LIN {X 0,Y 363.138,Z 659.015,A -85,B 0,C 180,E1 -13740.563,E2 -13740.563} C_VEL
LIN {X 0,Y 360.439,Z 673.892,A -85,B 0,C 180,E1 -13742.1,E2 -13742.1} C_VEL
LIN {X 0,Y 357.89,Z 687.3,A -85,B 0,C 180,E1 -13743.78,E2 -13743.78} C_VEL
LIN {X 0,Y 355.542,Z 698.752,A -85,B 0,C 180,E1 -13745.476,E2 -13745.476} C_VEL
LIN {X 0,Y 353.243,Z 710.279,A -85,B 0,C 180,E1 -13747.483,E2 -13747.483} C_VEL
LIN {X 0,Y 351.316,Z 720.192,A -85,B 0,C 180,E1 -13749.509,E2 -13749.509} C_VEL
LIN {X 0,Y 349.632,Z 729.753,A -85,B 0,C 180,E1 -13751.848,E2 -13751.848} C_VEL
LIN {X 0,Y 348.256,Z 737.796,A -85,B 0,C 180,E1 -13754.192,E2 -13754.192} C_VEL
LIN {X 0,Y 347.388,Z 744.678,A -85,B 0,C 180,E1 -13756.605,E2 -13756.605} C_VEL
LIN {X 0,Y 346.742,Z 750.015,A -85,B 0,C 180,E1 -13758.9,E2 -13758.9} C_VEL
LIN {X 0,Y 346.509,Z 753.412,A -85,B 0,C 180,E1 -13760.663,E2 -13760.663} C_VEL
LIN {X 0,Y 346.404,Z 757.9,A -85,B 0,C 180,E1 -13763.786,E2 -13763.786} C_VEL
LIN {X 0,Y 346.302,Z 760.292,A -85,B 0,C 180,E1 -13766.511,E2 -13766.511} C_VEL
LIN {X 0,Y 346.476,Z 761.273,A -85,B 0,C 180,E1 -13768.839,E2 -13768.839} C_VEL
LIN {X 0,Y 346.473,Z 761.269,A -85,B 0,C 180,E1 -13771.164,E2 -13771.164} C_VEL
LIN {X 0,Y 346.298,Z 760.218,A -85,B 0,C 180,E1 -13773.492,E2 -13773.492} C_VEL
LIN {X 0,Y 346.413,Z 758.208,A -85,B 0,C 180,E1 -13775.823,E2 -13775.823} C_VEL
LIN {X 0,Y 346.413,Z 755.082,A -85,B 0,C 180,E1 -13778.166,E2 -13778.166} C_VEL
LIN {X 0,Y 346.634,Z 750.942,A -85,B 0,C 180,E1 -13780.515,E2 -13780.515} C_VEL
LIN {X 0,Y 347.396,Z 744.256,A -85,B 0,C 180,E1 -13783.388,E2 -13783.388} C_VEL
LIN {X 0,Y 348.261,Z 737.113,A -85,B 0,C 180,E1 -13785.81,E2 -13785.81} C_VEL
LIN {X 0,Y 349.599,Z 728.749,A -85,B 0,C 180,E1 -13788.157,E2 -13788.157} C_VEL
LIN {X 0,Y 351.25,Z 718.757,A -85,B 0,C 180,E1 -13790.497,E2 -13790.497} C_VEL
LIN {X 0,Y 353.131,Z 708.481,A -85,B 0,C 180,E1 -13792.528,E2 -13792.528} C_VEL
LIN {X 0,Y 355.383,Z 696.336,A -85,B 0,C 180,E1 -13794.539,E2 -13794.539} C_VEL
LIN {X 0,Y 357.855,Z 682.977,A -85,B 0,C 180,E1 -13796.382,E2 -13796.382} C_VEL
LIN {X 0,Y 359.935,Z 670.909,A -85,B 0,C 180,E1 -13797.787,E2 -13797.787} C_VEL
LIN {X 0,Y 362.169,Z 656.954,A -85,B 0,C 180,E1 -13799.164,E2 -13799.164} C_VEL
LIN {X 0,Y 366.243,Z 636.712,A -85,B 0,C 180,E1 -13801.046,E2 -13801.046} C_VEL
LIN {X 0,Y 367.595,Z 629.602,A -85,B 0,C 180,E1 -13801.641,E2 -13801.641} C_VEL
LIN {X 0,Y 366.859,Z 616.235,A -85,B 0,C 180,E1 -13803.04,E2 -13803.04} C_VEL
LIN {X 0,Y 366.505,Z 599.284,A -85,B 0,C 180,E1 -13804.67,E2 -13804.67} C_VEL
LIN {X 0,Y 365.301,Z 587.346,A -85,B 0,C 180,E1 -13805.937,E2 -13805.937} C_VEL
LIN {X 0,Y 363.618,Z 576.417,A -85,B 0,C 180,E1 -13807.262,E2 -13807.262} C_VEL
LIN {X 0,Y 362.231,Z 569.674,A -85,B 0,C 180,E1 -13808.224,E2 -13808.224} C_VEL
LIN {X 0,Y 361.08,Z 564.227,A -85,B 0,C 180,E1 -13809.07,E2 -13809.07} C_VEL
LIN {X 0,Y 360.001,Z 559.824,A -85,B 0,C 180,E1 -13809.871,E2 -13809.871} C_VEL
LIN {X 0,Y 359.549,Z 557.218,A -85,B 0,C 180,E1 -13810.331,E2 -13810.331} C_VEL
LIN {X 0,Y 357.667,Z 548.632,A -85,B 0,C 180,E1 -13812.333,E2 -13812.333} C_VEL
LIN {X 0,Y 356.299,Z 544.697,A -85,B 0,C 180,E1 -13814.076,E2 -13814.076} C_VEL
LIN {X 0,Y 355.931,Z 542.529,A -85,B 0,C 180,E1 -13815.304,E2 -13815.304} C_VEL
LIN {X 0,Y 356.172,Z 540.509,A -85,B 0,C 180,E1 -13816.894,E2 -13816.894} C_VEL
LIN {X 0,Y 356.781,Z 539.56,A -85,B 0,C 180,E1 -13817.953,E2 -13817.953} C_VEL
LIN {X 0,Y 358.337,Z 540.28,A -85,B 0,C 180,E1 -13819.899,E2 -13819.899} C_VEL
LIN {X 0,Y 360.559,Z 541.255,A -85,B 0,C 180,E1 -13821.411,E2 -13821.411} C_VEL
LIN {X 0,Y 362.779,Z 542.718,A -85,B 0,C 180,E1 -13822.588,E2 -13822.588} C_VEL
LIN {X 0,Y 366.479,Z 546.75,A -85,B 0,C 180,E1 -13824.334,E2 -13824.334} C_VEL
LIN {X 0,Y 369.216,Z 550.249,A -85,B 0,C 180,E1 -13825.476,E2 -13825.476} C_VEL
LIN {X 0,Y 372.007,Z 554.619,A -85,B 0,C 180,E1 -13826.595,E2 -13826.595} C_VEL
LIN {X 0,Y 373.776,Z 559.648,A -85,B 0,C 180,E1 -13827.486,E2 -13827.486} C_VEL
LIN {X 0,Y 374.288,Z 561.573,A -85,B 0,C 180,E1 -13827.801,E2 -13827.801} C_VEL
LIN {X 0,Y 373.296,Z 567.896,A -85,B 0,C 180,E1 -13828.306,E2 -13828.306} C_VEL
LIN {X 0,Y 370.01,Z 584.666,A -85,B 0,C 180,E1 -13829.779,E2 -13829.779} C_VEL
LIN {X 0,Y 366.898,Z 599.707,A -85,B 0,C 180,E1 -13831.388,E2 -13831.388} C_VEL
LIN {X 0,Y 363.907,Z 613.147,A -85,B 0,C 180,E1 -13833.09,E2 -13833.09} C_VEL
LIN {X 0,Y 360.966,Z 625.629,A -85,B 0,C 180,E1 -13834.947,E2 -13834.947} C_VEL
LIN {X 0,Y 358.09,Z 637.94,A -85,B 0,C 180,E1 -13837.15,E2 -13837.15} C_VEL
LIN {X 0,Y 355.396,Z 648.703,A -85,B 0,C 180,E1 -13839.451,E2 -13839.451} C_VEL
LIN {X 0,Y 353.515,Z 656.559,A -85,B 0,C 180,E1 -13841.453,E2 -13841.453} C_VEL
LIN {X 0,Y 351.734,Z 664.142,A -85,B 0,C 180,E1 -13843.756,E2 -13843.756} C_VEL
LIN {X 0,Y 350.191,Z 670.343,A -85,B 0,C 180,E1 -13846.065,E2 -13846.065} C_VEL
LIN {X 0,Y 349.135,Z 675.359,A -85,B 0,C 180,E1 -13848.388,E2 -13848.388} C_VEL
LIN {X 0,Y 348.342,Z 679.303,A -85,B 0,C 180,E1 -13850.712,E2 -13850.712} C_VEL
LIN {X 0,Y 347.779,Z 682.101,A -85,B 0,C 180,E1 -13853.036,E2 -13853.036} C_VEL
LIN {X 0,Y 347.335,Z 683.994,A -85,B 0,C 180,E1 -13855.358,E2 -13855.358} C_VEL
LIN {X 0,Y 346.936,Z 684.871,A -85,B 0,C 180,E1 -13857.679,E2 -13857.679} C_VEL
LIN {X 0,Y 346.757,Z 684.777,A -85,B 0,C 180,E1 -13860.001,E2 -13860.001} C_VEL
LIN {X 0,Y 346.897,Z 683.694,A -85,B 0,C 180,E1 -13862.323,E2 -13862.323} C_VEL
LIN {X 0,Y 347.092,Z 681.603,A -85,B 0,C 180,E1 -13864.646,E2 -13864.646} C_VEL
LIN {X 0,Y 347.314,Z 678.062,A -85,B 0,C 180,E1 -13867.276,E2 -13867.276} C_VEL
LIN {X 0,Y 347.759,Z 673.198,A -85,B 0,C 180,E1 -13869.892,E2 -13869.892} C_VEL
LIN {X 0,Y 348.3,Z 667.576,A -85,B 0,C 180,E1 -13872.232,E2 -13872.232} C_VEL
LIN {X 0,Y 349.313,Z 660.704,A -85,B 0,C 180,E1 -13874.566,E2 -13874.566} C_VEL
LIN {X 0,Y 350.473,Z 652.438,A -85,B 0,C 180,E1 -13876.904,E2 -13876.904} C_VEL
LIN {X 0,Y 352.043,Z 642.556,A -85,B 0,C 180,E1 -13879.233,E2 -13879.233} C_VEL
LIN {X 0,Y 353.675,Z 632.321,A -85,B 0,C 180,E1 -13881.264,E2 -13881.264} C_VEL
LIN {X 0,Y 355.6,Z 620.344,A -85,B 0,C 180,E1 -13883.284,E2 -13883.284} C_VEL
LIN {X 0,Y 357.692,Z 607.625,A -85,B 0,C 180,E1 -13885.097,E2 -13885.097} C_VEL
LIN {X 0,Y 359.886,Z 593.111,A -85,B 0,C 180,E1 -13886.847,E2 -13886.847} C_VEL
LIN {X 0,Y 361.871,Z 579.208,A -85,B 0,C 180,E1 -13888.255,E2 -13888.255} C_VEL
LIN {X 0,Y 363.664,Z 565.161,A -85,B 0,C 180,E1 -13889.457,E2 -13889.457} C_VEL
LIN {X 0,Y 364.728,Z 556.813,A -85,B 0,C 180,E1 -13890.067,E2 -13890.067} C_VEL
LIN {X 0,Y 364.326,Z 554.698,A -85,B 0,C 180,E1 -13890.261,E2 -13890.261} C_VEL
LIN {X 0,Y 358.467,Z 539.997,A -85,B 0,C 180,E1 -13891.771,E2 -13891.771} C_VEL
LIN {X 0,Y 351.64,Z 524.321,A -85,B 0,C 180,E1 -13893.255,E2 -13893.255} C_VEL
LIN {X 0,Y 347.929,Z 516.364,A -85,B 0,C 180,E1 -13893.96,E2 -13893.96} C_VEL
LIN {X 0,Y 347.754,Z 515.48,A -85,B 0,C 180,E1 -13894.044,E2 -13894.044} C_VEL
LIN {X 0,Y 347.771,Z 515.479,A -85,B 0,C 180,E1 -13897.32,E2 -13897.32} C_VEL
LIN {X 0,Y 347.738,Z 515.483,A -85,B 0,C 180,E1 -13900.297,E2 -13900.297} C_VEL
LIN {X 0,Y 347.729,Z 515.483,A -85,B 0,C 180,E1 -13903.408,E2 -13903.408} C_VEL
LIN {X 0,Y 347.731,Z 515.482,A -85,B 0,C 180,E1 -13906.686,E2 -13906.686} C_VEL
LIN {X 0,Y 347.753,Z 515.482,A -85,B 0,C 180,E1 -13910.173,E2 -13910.173} C_VEL
LIN {X 0,Y 347.768,Z 515.478,A -85,B 0,C 180,E1 -13912.679,E2 -13912.679} C_VEL
LIN {X 0,Y 347.754,Z 515.485,A -85,B 0,C 180,E1 -13915.956,E2 -13915.956} C_VEL
LIN {X 0,Y 347.831,Z 515.679,A -85,B 0,C 180,E1 -13919.659,E2 -13919.659} C_VEL
LIN {X 0,Y 348.651,Z 519.993,A -85,B 0,C 180,E1 -13922.492,E2 -13922.492} C_VEL
LIN {X 0,Y 349.099,Z 524.824,A -85,B 0,C 180,E1 -13925.624,E2 -13925.624} C_VEL
LIN {X 0,Y 349.014,Z 529.788,A -85,B 0,C 180,E1 -13928.748,E2 -13928.748} C_VEL
LIN {X 0,Y 348.958,Z 531.353,A -85,B 0,C 180,E1 -13929.737,E2 -13929.737} C_VEL
LIN {X 0,Y 350.286,Z 534.706,A -85,B 0,C 180,E1 -13929.954,E2 -13929.954} C_VEL
LIN {X 0,Y 357.426,Z 551.292,A -85,B 0,C 180,E1 -13931.148,E2 -13931.148} C_VEL
LIN {X 0,Y 362.757,Z 565.923,A -85,B 0,C 180,E1 -13932.276,E2 -13932.276} C_VEL
LIN {X 0,Y 366.78,Z 578.552,A -85,B 0,C 180,E1 -13933.351,E2 -13933.351} C_VEL
LIN {X 0,Y 367.752,Z 582.268,A -85,B 0,C 180,E1 -13933.67,E2 -13933.67} C_VEL
LIN {X 0,Y 366.186,Z 596.258,A -85,B 0,C 180,E1 -13934.555,E2 -13934.555} C_VEL
LIN {X 0,Y 364.346,Z 610.122,A -85,B 0,C 180,E1 -13935.619,E2 -13935.619} C_VEL
LIN {X 0,Y 362.201,Z 624.446,A -85,B 0,C 180,E1 -13936.963,E2 -13936.963} C_VEL
LIN {X 0,Y 359.939,Z 637.66,A -85,B 0,C 180,E1 -13938.454,E2 -13938.454} C_VEL
LIN {X 0,Y 357.75,Z 649.93,A -85,B 0,C 180,E1 -13940.101,E2 -13940.101} C_VEL
LIN {X 0,Y 355.43,Z 662.146,A -85,B 0,C 180,E1 -13942.043,E2 -13942.043} C_VEL
LIN {X 0,Y 353.434,Z 672.571,A -85,B 0,C 180,E1 -13944.006,E2 -13944.006} C_VEL
LIN {X 0,Y 351.459,Z 682.629,A -85,B 0,C 180,E1 -13946.273,E2 -13946.273} C_VEL
LIN {X 0,Y 349.96,Z 690.122,A -85,B 0,C 180,E1 -13948.273,E2 -13948.273} C_VEL
LIN {X 0,Y 348.726,Z 697.402,A -85,B 0,C 180,E1 -13950.576,E2 -13950.576} C_VEL
LIN {X 0,Y 347.732,Z 703.363,A -85,B 0,C 180,E1 -13952.895,E2 -13952.895} C_VEL
LIN {X 0,Y 347.128,Z 708.203,A -85,B 0,C 180,E1 -13955.226,E2 -13955.226} C_VEL
LIN {X 0,Y 346.793,Z 711.131,A -85,B 0,C 180,E1 -13956.983,E2 -13956.983} C_VEL
LIN {X 0,Y 346.41,Z 714.204,A -85,B 0,C 180,E1 -13959.339,E2 -13959.339} C_VEL
LIN {X 0,Y 346.25,Z 716.196,A -85,B 0,C 180,E1 -13961.71,E2 -13961.71} C_VEL
LIN {X 0,Y 346.106,Z 717.28,A -85,B 0,C 180,E1 -13964.102,E2 -13964.102} C_VEL
LIN {X 0,Y 346.124,Z 717.343,A -85,B 0,C 180,E1 -13966.514,E2 -13966.514} C_VEL
LIN {X 0,Y 346.211,Z 716.409,A -85,B 0,C 180,E1 -13968.952,E2 -13968.952} C_VEL
LIN {X 0,Y 346.534,Z 714.459,A -85,B 0,C 180,E1 -13971.409,E2 -13971.409} C_VEL
LIN {X 0,Y 347.15,Z 710.676,A -85,B 0,C 180,E1 -13974.352,E2 -13974.352} C_VEL
LIN {X 0,Y 347.792,Z 707.099,A -85,B 0,C 180,E1 -13976.394,E2 -13976.394} C_VEL
LIN {X 0,Y 348.818,Z 701.582,A -85,B 0,C 180,E1 -13978.916,E2 -13978.916} C_VEL
LIN {X 0,Y 350.217,Z 694.579,A -85,B 0,C 180,E1 -13981.448,E2 -13981.448} C_VEL
LIN {X 0,Y 351.089,Z 690.641,A -85,B 0,C 180,E1 -13982.667,E2 -13982.667} C_VEL
LIN {X 0,Y 351.095,Z 687.889,A -85,B 0,C 180,E1 -13983.52,E2 -13983.52} C_VEL
LIN {X 0,Y 348.004,Z 678.593,A -85,B 0,C 180,E1 -13986.342,E2 -13986.342} C_VEL
LIN {X 0,Y 348.214,Z 675.241,A -85,B 0,C 180,E1 -13987.147,E2 -13987.147} C_VEL
LIN {X 0,Y 350.67,Z 665.25,A -85,B 0,C 180,E1 -13989.145,E2 -13989.145} C_VEL
LIN {X 0,Y 353.23,Z 654.18,A -85,B 0,C 180,E1 -13991.037,E2 -13991.037} C_VEL
LIN {X 0,Y 355.96,Z 642.094,A -85,B 0,C 180,E1 -13992.774,E2 -13992.774} C_VEL
LIN {X 0,Y 358.839,Z 628.158,A -85,B 0,C 180,E1 -13994.439,E2 -13994.439} C_VEL
LIN {X 0,Y 361.392,Z 614.482,A -85,B 0,C 180,E1 -13995.789,E2 -13995.789} C_VEL
LIN {X 0,Y 363.625,Z 600.382,A -85,B 0,C 180,E1 -13996.953,E2 -13996.953} C_VEL
LIN {X 0,Y 365.568,Z 586.338,A -85,B 0,C 180,E1 -13997.896,E2 -13997.896} C_VEL
LIN {X 0,Y 362.056,Z 574.059,A -85,B 0,C 180,E1 -13999.17,E2 -13999.17} C_VEL
LIN {X 0,Y 356.721,Z 560.139,A -85,B 0,C 180,E1 -14000.647,E2 -14000.647} C_VEL
LIN {X 0,Y 351.009,Z 548.123,A -85,B 0,C 180,E1 -14001.941,E2 -14001.941} C_VEL
LIN {X 0,Y 345.13,Z 537.197,A -85,B 0,C 180,E1 -14003.156,E2 -14003.156} C_VEL
LIN {X 0,Y 343.491,Z 534.071,A -85,B 0,C 180,E1 -14003.498,E2 -14003.498} C_VEL
LIN {X 0,Y 343.298,Z 533.359,A -85,B 0,C 180,E1 -14003.58,E2 -14003.58} C_VEL
LIN {X 0,Y 343.138,Z 529.364,A -85,B 0,C 180,E1 -14006.426,E2 -14006.426} C_VEL
LIN {X 0,Y 342.502,Z 525.206,A -85,B 0,C 180,E1 -14009.518,E2 -14009.518} C_VEL
LIN {X 0,Y 341.673,Z 520.486,A -85,B 0,C 180,E1 -14013.093,E2 -14013.093} C_VEL
LIN {X 0,Y 340.75,Z 516.352,A -85,B 0,C 180,E1 -14016.325,E2 -14016.325} C_VEL
LIN {X 0,Y 340.757,Z 516.352,A -85,B 0,C 180,E1 -14019.474,E2 -14019.474} C_VEL
LIN {X 0,Y 340.849,Z 516.341,A -85,B 0,C 180,E1 -14021.983,E2 -14021.983} C_VEL
LIN {X 0,Y 340.86,Z 516.334,A -85,B 0,C 180,E1 -14025.704,E2 -14025.704} C_VEL
LIN {X 0,Y 340.865,Z 516.331,A -85,B 0,C 180,E1 -14029.305,E2 -14029.305} C_VEL
LIN {X 0,Y 341.068,Z 516.31,A -85,B 0,C 180,E1 -14032.898,E2 -14032.898} C_VEL
LIN {X 0,Y 341.161,Z 516.296,A -85,B 0,C 180,E1 -14037.638,E2 -14037.638} C_VEL
LIN {X 0,Y 341.307,Z 516.284,A -85,B 0,C 180,E1 -14039.999,E2 -14039.999} C_VEL
LIN {X 0,Y 341.16,Z 516.293,A -85,B 0,C 180,E1 -14042.361,E2 -14042.361} C_VEL
LIN {X 0,Y 341.064,Z 516.312,A -85,B 0,C 180,E1 -14047.101,E2 -14047.101} C_VEL
LIN {X 0,Y 340.865,Z 516.337,A -85,B 0,C 180,E1 -14050.693,E2 -14050.693} C_VEL
LIN {X 0,Y 340.852,Z 516.339,A -85,B 0,C 180,E1 -14054.325,E2 -14054.325} C_VEL
LIN {X 0,Y 340.828,Z 516.3,A -85,B 0,C 180,E1 -14058.468,E2 -14058.468} C_VEL
LIN {X 0,Y 340.769,Z 516.347,A -85,B 0,C 180,E1 -14061.868,E2 -14061.868} C_VEL
LIN {X 0,Y 340.766,Z 516.315,A -85,B 0,C 180,E1 -14065.664,E2 -14065.664} C_VEL
LIN {X 0,Y 340.732,Z 516.355,A -85,B 0,C 180,E1 -14068.32,E2 -14068.32} C_VEL
LIN {X 0,Y 340.694,Z 516.359,A -85,B 0,C 180,E1 -14071.044,E2 -14071.044} C_VEL
LIN {X 0,Y 340.708,Z 516.454,A -85,B 0,C 180,E1 -14072.959,E2 -14072.959} C_VEL
LIN {X 0,Y 342.386,Z 523.899,A -85,B 0,C 180,E1 -14076.531,E2 -14076.531} C_VEL
LIN {X 0,Y 344.124,Z 531.611,A -85,B 0,C 180,E1 -14080.039,E2 -14080.039} C_VEL
LIN {X 0,Y 346.146,Z 541.37,A -85,B 0,C 180,E1 -14084.227,E2 -14084.227} C_VEL
LIN {X 0,Y 347.726,Z 549.268,A -85,B 0,C 180,E1 -14087.44,E2 -14087.44} C_VEL
LIN {X 0,Y 347.671,Z 553.507,A -85,B 0,C 180,E1 -14089.035,E2 -14089.035} C_VEL
LIN {X 0,Y 346.408,Z 563.412,A -85,B 0,C 180,E1 -14092.575,E2 -14092.575} C_VEL
LIN {X 0,Y 347.388,Z 567.065,A -85,B 0,C 180,E1 -14092.816,E2 -14092.816} C_VEL
LIN {X 0,Y 352.342,Z 581.881,A -85,B 0,C 180,E1 -14093.927,E2 -14093.927} C_VEL
LIN {X 0,Y 355.976,Z 596.537,A -85,B 0,C 180,E1 -14094.969,E2 -14094.969} C_VEL
LIN {X 0,Y 359.262,Z 613.763,A -85,B 0,C 180,E1 -14096.296,E2 -14096.296} C_VEL
LIN {X 0,Y 361.544,Z 630.3,A -85,B 0,C 180,E1 -14097.719,E2 -14097.719} C_VEL
LIN {X 0,Y 360.072,Z 641.655,A -85,B 0,C 180,E1 -14098.528,E2 -14098.528} C_VEL
LIN {X 0,Y 357.47,Z 656.478,A -85,B 0,C 180,E1 -14099.748,E2 -14099.748} C_VEL
LIN {X 0,Y 354.912,Z 670.176,A -85,B 0,C 180,E1 -14101.141,E2 -14101.141} C_VEL
LIN {X 0,Y 352.269,Z 683.008,A -85,B 0,C 180,E1 -14102.688,E2 -14102.688} C_VEL
LIN {X 0,Y 349.749,Z 695.417,A -85,B 0,C 180,E1 -14104.469,E2 -14104.469} C_VEL
LIN {X 0,Y 347.272,Z 707.025,A -85,B 0,C 180,E1 -14106.443,E2 -14106.443} C_VEL
LIN {X 0,Y 344.833,Z 718.604,A -85,B 0,C 180,E1 -14108.793,E2 -14108.793} C_VEL
LIN {X 0,Y 342.955,Z 728.348,A -85,B 0,C 180,E1 -14111.172,E2 -14111.172} C_VEL
LIN {X 0,Y 341.636,Z 735.634,A -85,B 0,C 180,E1 -14113.263,E2 -14113.263} C_VEL
LIN {X 0,Y 340.511,Z 743.379,A -85,B 0,C 180,E1 -14115.942,E2 -14115.942} C_VEL
LIN {X 0,Y 339.709,Z 749.641,A -85,B 0,C 180,E1 -14118.667,E2 -14118.667} C_VEL
LIN {X 0,Y 339.423,Z 753.021,A -85,B 0,C 180,E1 -14120.467,E2 -14120.467} C_VEL
LIN {X 0,Y 339.318,Z 756.502,A -85,B 0,C 180,E1 -14122.863,E2 -14122.863} C_VEL
LIN {X 0,Y 339.224,Z 759.021,A -85,B 0,C 180,E1 -14125.248,E2 -14125.248} C_VEL
LIN {X 0,Y 339.296,Z 760.457,A -85,B 0,C 180,E1 -14127.627,E2 -14127.627} C_VEL
LIN {X 0,Y 339.38,Z 760.964,A -85,B 0,C 180,E1 -14130.001,E2 -14130.001} C_VEL
LIN {X 0,Y 339.368,Z 760.397,A -85,B 0,C 180,E1 -14132.375,E2 -14132.375} C_VEL
LIN {X 0,Y 339.297,Z 758.874,A -85,B 0,C 180,E1 -14134.754,E2 -14134.754} C_VEL
LIN {X 0,Y 339.322,Z 756.269,A -85,B 0,C 180,E1 -14137.14,E2 -14137.14} C_VEL
LIN {X 0,Y 339.516,Z 751.522,A -85,B 0,C 180,E1 -14140.135,E2 -14140.135} C_VEL
LIN {X 0,Y 340.014,Z 746.466,A -85,B 0,C 180,E1 -14142.536,E2 -14142.536} C_VEL
LIN {X 0,Y 340.793,Z 740.198,A -85,B 0,C 180,E1 -14144.94,E2 -14144.94} C_VEL
LIN {X 0,Y 342.192,Z 731.492,A -85,B 0,C 180,E1 -14147.635,E2 -14147.635} C_VEL
LIN {X 0,Y 343.646,Z 722.545,A -85,B 0,C 180,E1 -14149.916,E2 -14149.916} C_VEL
LIN {X 0,Y 345.555,Z 712.361,A -85,B 0,C 180,E1 -14152.103,E2 -14152.103} C_VEL
LIN {X 0,Y 347.73,Z 701.327,A -85,B 0,C 180,E1 -14154.108,E2 -14154.108} C_VEL
LIN {X 0,Y 350.187,Z 688.648,A -85,B 0,C 180,E1 -14156.042,E2 -14156.042} C_VEL
LIN {X 0,Y 352.588,Z 675.091,A -85,B 0,C 180,E1 -14157.771,E2 -14157.771} C_VEL
LIN {X 0,Y 358.329,Z 646.316,A -85,B 0,C 180,E1 -14160.825,E2 -14160.825} C_VEL
LIN {X 0,Y 361.546,Z 630.746,A -85,B 0,C 180,E1 -14162.238,E2 -14162.238} C_VEL
LIN {X 0,Y 361.175,Z 617.764,A -85,B 0,C 180,E1 -14163.682,E2 -14163.682} C_VEL
LIN {X 0,Y 361.208,Z 601.756,A -85,B 0,C 180,E1 -14165.305,E2 -14165.305} C_VEL
LIN {X 0,Y 360.189,Z 588.151,A -85,B 0,C 180,E1 -14166.871,E2 -14166.871} C_VEL
LIN {X 0,Y 358.894,Z 578.855,A -85,B 0,C 180,E1 -14168.119,E2 -14168.119} C_VEL
LIN {X 0,Y 357.589,Z 570.516,A -85,B 0,C 180,E1 -14169.394,E2 -14169.394} C_VEL
LIN {X 0,Y 356.104,Z 562.093,A -85,B 0,C 180,E1 -14170.975,E2 -14170.975} C_VEL
LIN {X 0,Y 354.792,Z 554.339,A -85,B 0,C 180,E1 -14172.869,E2 -14172.869} C_VEL
LIN {X 0,Y 353.854,Z 551.132,A -85,B 0,C 180,E1 -14174.357,E2 -14174.357} C_VEL
LIN {X 0,Y 353.602,Z 548.557,A -85,B 0,C 180,E1 -14175.922,E2 -14175.922} C_VEL
LIN {X 0,Y 354.197,Z 546.683,A -85,B 0,C 180,E1 -14177.575,E2 -14177.575} C_VEL
LIN {X 0,Y 355.294,Z 546.707,A -85,B 0,C 180,E1 -14179.25,E2 -14179.25} C_VEL
LIN {X 0,Y 357.482,Z 547.514,A -85,B 0,C 180,E1 -14181.016,E2 -14181.016} C_VEL
LIN {X 0,Y 360.833,Z 550.296,A -85,B 0,C 180,E1 -14182.994,E2 -14182.994} C_VEL
LIN {X 0,Y 364.195,Z 554.214,A -85,B 0,C 180,E1 -14184.626,E2 -14184.626} C_VEL
LIN {X 0,Y 367.18,Z 558.764,A -85,B 0,C 180,E1 -14185.983,E2 -14185.983} C_VEL
LIN {X 0,Y 368.459,Z 561.71,A -85,B 0,C 180,E1 -14186.619,E2 -14186.619} C_VEL
LIN {X 0,Y 369.265,Z 565.365,A -85,B 0,C 180,E1 -14187.23,E2 -14187.23} C_VEL
LIN {X 0,Y 366.059,Z 580.597,A -85,B 0,C 180,E1 -14188.527,E2 -14188.527} C_VEL
LIN {X 0,Y 363.01,Z 594.419,A -85,B 0,C 180,E1 -14189.938,E2 -14189.938} C_VEL
LIN {X 0,Y 359.858,Z 607.979,A -85,B 0,C 180,E1 -14191.563,E2 -14191.563} C_VEL
LIN {X 0,Y 356.657,Z 620.811,A -85,B 0,C 180,E1 -14193.366,E2 -14193.366} C_VEL
LIN {X 0,Y 353.659,Z 632.613,A -85,B 0,C 180,E1 -14195.335,E2 -14195.335} C_VEL
LIN {X 0,Y 350.638,Z 644.102,A -85,B 0,C 180,E1 -14197.616,E2 -14197.616} C_VEL
LIN {X 0,Y 348.377,Z 652.718,A -85,B 0,C 180,E1 -14199.636,E2 -14199.636} C_VEL
LIN {X 0,Y 346.434,Z 660.061,A -85,B 0,C 180,E1 -14201.673,E2 -14201.673} C_VEL
LIN {X 0,Y 344.609,Z 667.128,A -85,B 0,C 180,E1 -14204.019,E2 -14204.019} C_VEL
LIN {X 0,Y 343.079,Z 672.996,A -85,B 0,C 180,E1 -14206.375,E2 -14206.375} C_VEL
LIN {X 0,Y 342.019,Z 677.625,A -85,B 0,C 180,E1 -14208.743,E2 -14208.743} C_VEL
LIN {X 0,Y 341.2,Z 681.494,A -85,B 0,C 180,E1 -14211.381,E2 -14211.381} C_VEL
LIN {X 0,Y 340.473,Z 684.179,A -85,B 0,C 180,E1 -14214.077,E2 -14214.077} C_VEL
LIN {X 0,Y 340.089,Z 685.513,A -85,B 0,C 180,E1 -14216.446,E2 -14216.446} C_VEL
LIN {X 0,Y 339.774,Z 685.809,A -85,B 0,C 180,E1 -14218.815,E2 -14218.815} C_VEL
LIN {X 0,Y 339.73,Z 685.179,A -85,B 0,C 180,E1 -14221.186,E2 -14221.186} C_VEL
LIN {X 0,Y 340.043,Z 683.494,A -85,B 0,C 180,E1 -14223.555,E2 -14223.555} C_VEL
LIN {X 0,Y 340.063,Z 680.87,A -85,B 0,C 180,E1 -14225.932,E2 -14225.932} C_VEL
LIN {X 0,Y 340.432,Z 677.2,A -85,B 0,C 180,E1 -14228.309,E2 -14228.309} C_VEL
LIN {X 0,Y 340.859,Z 672.382,A -85,B 0,C 180,E1 -14230.695,E2 -14230.695} C_VEL
LIN {X 0,Y 341.543,Z 666.42,A -85,B 0,C 180,E1 -14233.083,E2 -14233.083} C_VEL
LIN {X 0,Y 342.673,Z 659.135,A -85,B 0,C 180,E1 -14235.464,E2 -14235.464} C_VEL
LIN {X 0,Y 344.013,Z 650.33,A -85,B 0,C 180,E1 -14237.845,E2 -14237.845} C_VEL
LIN {X 0,Y 345.511,Z 641.257,A -85,B 0,C 180,E1 -14239.921,E2 -14239.921} C_VEL
LIN {X 0,Y 347.24,Z 630.713,A -85,B 0,C 180,E1 -14241.99,E2 -14241.99} C_VEL
LIN {X 0,Y 349.372,Z 618.351,A -85,B 0,C 180,E1 -14244.039,E2 -14244.039} C_VEL
LIN {X 0,Y 351.54,Z 605.148,A -85,B 0,C 180,E1 -14245.888,E2 -14245.888} C_VEL
LIN {X 0,Y 353.888,Z 590.046,A -85,B 0,C 180,E1 -14247.66,E2 -14247.66} C_VEL
LIN {X 0,Y 356.019,Z 575.397,A -85,B 0,C 180,E1 -14249.086,E2 -14249.086} C_VEL
LIN {X 0,Y 357.824,Z 560.818,A -85,B 0,C 180,E1 -14250.279,E2 -14250.279} C_VEL
LIN {X 0,Y 358.164,Z 558.328,A -85,B 0,C 180,E1 -14250.462,E2 -14250.462} C_VEL
LIN {X 0,Y 353.964,Z 546.899,A -85,B 0,C 180,E1 -14251.682,E2 -14251.682} C_VEL
LIN {X 0,Y 347.166,Z 530.919,A -85,B 0,C 180,E1 -14253.29,E2 -14253.29} C_VEL
LIN {X 0,Y 340.877,Z 517.276,A -85,B 0,C 180,E1 -14254.565,E2 -14254.565} C_VEL
LIN {X 0,Y 340.718,Z 516.359,A -85,B 0,C 180,E1 -14254.65,E2 -14254.65} C_VEL
LIN {X 0,Y 340.717,Z 516.356,A -85,B 0,C 180,E1 -14258.386,E2 -14258.386} C_VEL
LIN {X 0,Y 340.704,Z 516.359,A -85,B 0,C 180,E1 -14262.045,E2 -14262.045} C_VEL
LIN {X 0,Y 340.657,Z 516.365,A -85,B 0,C 180,E1 -14266.227,E2 -14266.227} C_VEL
LIN {X 0,Y 340.694,Z 516.36,A -85,B 0,C 180,E1 -14269.753,E2 -14269.753} C_VEL
LIN {X 0,Y 340.711,Z 516.357,A -85,B 0,C 180,E1 -14273.258,E2 -14273.258} C_VEL
LIN {X 0,Y 340.698,Z 516.365,A -85,B 0,C 180,E1 -14276.153,E2 -14276.153} C_VEL
LIN {X 0,Y 340.763,Z 516.532,A -85,B 0,C 180,E1 -14279.102,E2 -14279.102} C_VEL
LIN {X 0,Y 341.665,Z 521.168,A -85,B 0,C 180,E1 -14282.192,E2 -14282.192} C_VEL
LIN {X 0,Y 342.082,Z 524.974,A -85,B 0,C 180,E1 -14284.686,E2 -14284.686} C_VEL
LIN {X 0,Y 342.113,Z 529.503,A -85,B 0,C 180,E1 -14287.584,E2 -14287.584} C_VEL
LIN {X 0,Y 342.064,Z 531.756,A -85,B 0,C 180,E1 -14289.014,E2 -14289.014} C_VEL
LIN {X 0,Y 343.433,Z 535.172,A -85,B 0,C 180,E1 -14289.256,E2 -14289.256} C_VEL
LIN {X 0,Y 350.584,Z 551.695,A -85,B 0,C 180,E1 -14290.488,E2 -14290.488} C_VEL
LIN {X 0,Y 355.695,Z 565.542,A -85,B 0,C 180,E1 -14291.594,E2 -14291.594} C_VEL
LIN {X 0,Y 360.053,Z 578.984,A -85,B 0,C 180,E1 -14292.767,E2 -14292.767} C_VEL
LIN {X 0,Y 361.397,Z 583.652,A -85,B 0,C 180,E1 -14293.19,E2 -14293.19} C_VEL
LIN {X 0,Y 359.755,Z 597.908,A -85,B 0,C 180,E1 -14294.126,E2 -14294.126} C_VEL
LIN {X 0,Y 357.64,Z 613.036,A -85,B 0,C 180,E1 -14295.343,E2 -14295.343} C_VEL
LIN {X 0,Y 355.441,Z 626.988,A -85,B 0,C 180,E1 -14296.71,E2 -14296.71} C_VEL
LIN {X 0,Y 353.081,Z 639.967,A -85,B 0,C 180,E1 -14298.227,E2 -14298.227} C_VEL
LIN {X 0,Y 350.874,Z 651.931,A -85,B 0,C 180,E1 -14299.905,E2 -14299.905} C_VEL
LIN {X 0,Y 348.5,Z 663.904,A -85,B 0,C 180,E1 -14301.884,E2 -14301.884} C_VEL
LIN {X 0,Y 346.437,Z 674.197,A -85,B 0,C 180,E1 -14303.898,E2 -14303.898} C_VEL
LIN {X 0,Y 344.444,Z 684.073,A -85,B 0,C 180,E1 -14306.197,E2 -14306.197} C_VEL
LIN {X 0,Y 342.916,Z 691.396,A -85,B 0,C 180,E1 -14308.237,E2 -14308.237} C_VEL
LIN {X 0,Y 341.643,Z 698.514,A -85,B 0,C 180,E1 -14310.588,E2 -14310.588} C_VEL
LIN {X 0,Y 340.653,Z 704.399,A -85,B 0,C 180,E1 -14312.955,E2 -14312.955} C_VEL
LIN {X 0,Y 340.015,Z 709.096,A -85,B 0,C 180,E1 -14315.336,E2 -14315.336} C_VEL
LIN {X 0,Y 339.698,Z 711.954,A -85,B 0,C 180,E1 -14317.129,E2 -14317.129} C_VEL
LIN {X 0,Y 339.289,Z 714.894,A -85,B 0,C 180,E1 -14319.537,E2 -14319.537} C_VEL
LIN {X 0,Y 339.147,Z 716.821,A -85,B 0,C 180,E1 -14321.958,E2 -14321.958} C_VEL
LIN {X 0,Y 339.027,Z 717.769,A -85,B 0,C 180,E1 -14324.403,E2 -14324.403} C_VEL
LIN {X 0,Y 339.05,Z 717.769,A -85,B 0,C 180,E1 -14326.868,E2 -14326.868} C_VEL
LIN {X 0,Y 339.186,Z 716.695,A -85,B 0,C 180,E1 -14329.36,E2 -14329.36} C_VEL
LIN {X 0,Y 339.523,Z 714.641,A -85,B 0,C 180,E1 -14331.874,E2 -14331.874} C_VEL
LIN {X 0,Y 340.164,Z 711.113,A -85,B 0,C 180,E1 -14334.622,E2 -14334.622} C_VEL
LIN {X 0,Y 340.95,Z 707.01,A -85,B 0,C 180,E1 -14336.966,E2 -14336.966} C_VEL
LIN {X 0,Y 342.073,Z 701.349,A -85,B 0,C 180,E1 -14339.542,E2 -14339.542} C_VEL
LIN {X 0,Y 343.641,Z 694.244,A -85,B 0,C 180,E1 -14342.121,E2 -14342.121} C_VEL
LIN {X 0,Y 345.741,Z 685.467,A -85,B 0,C 180,E1 -14344.69,E2 -14344.69} C_VEL
LIN {X 0,Y 348.214,Z 675.241,A -85,B 0,C 180,E1 -14347.147,E2 -14347.147} C_VEL
LIN {X 0,Y 348.455,Z 671.831,A -85,B 0,C 180,E1 -14347.941,E2 -14347.941} C_VEL
LIN {X 0,Y 346.114,Z 660.483,A -85,B 0,C 180,E1 -14350.593,E2 -14350.593} C_VEL
LIN {X 0,Y 346.557,Z 656.521,A -85,B 0,C 180,E1 -14351.318,E2 -14351.318} C_VEL
LIN {X 0,Y 349.466,Z 644.29,A -85,B 0,C 180,E1 -14353.136,E2 -14353.136} C_VEL
LIN {X 0,Y 352.458,Z 630.465,A -85,B 0,C 180,E1 -14354.857,E2 -14354.857} C_VEL
LIN {X 0,Y 355.368,Z 615.865,A -85,B 0,C 180,E1 -14356.348,E2 -14356.348} C_VEL
LIN {X 0,Y 357.587,Z 602.695,A -85,B 0,C 180,E1 -14357.476,E2 -14357.476} C_VEL
LIN {X 0,Y 359.609,Z 587.963,A -85,B 0,C 180,E1 -14358.507,E2 -14358.507} C_VEL
LIN {X 0,Y 355.396,Z 573.834,A -85,B 0,C 180,E1 -14360.053,E2 -14360.053} C_VEL
LIN {X 0,Y 350.055,Z 560.252,A -85,B 0,C 180,E1 -14361.571,E2 -14361.571} C_VEL
LIN {X 0,Y 342.993,Z 545.87,A -85,B 0,C 180,E1 -14363.215,E2 -14363.215} C_VEL
LIN {X 0,Y 338.639,Z 538.042,A -85,B 0,C 180,E1 -14364.151,E2 -14364.151} C_VEL
LIN {X 0,Y 336.883,Z 535.201,A -85,B 0,C 180,E1 -14364.521,E2 -14364.521} C_VEL
LIN {X 0,Y 336.469,Z 533.841,A -85,B 0,C 180,E1 -14364.667,E2 -14364.667} C_VEL
LIN {X 0,Y 336.252,Z 530.568,A -85,B 0,C 180,E1 -14367.082,E2 -14367.082} C_VEL
LIN {X 0,Y 335.68,Z 526.957,A -85,B 0,C 180,E1 -14369.835,E2 -14369.835} C_VEL
LIN {X 0,Y 335.065,Z 523.467,A -85,B 0,C 180,E1 -14372.519,E2 -14372.519} C_VEL
LIN {X 0,Y 334.412,Z 520.133,A -85,B 0,C 180,E1 -14375.145,E2 -14375.145} C_VEL
LIN {X 0,Y 333.679,Z 517.235,A -85,B 0,C 180,E1 -14377.557,E2 -14377.557} C_VEL
LIN {X 0,Y 333.786,Z 517.217,A -85,B 0,C 180,E1 -14381.588,E2 -14381.588} C_VEL
LIN {X 0,Y 333.799,Z 517.214,A -85,B 0,C 180,E1 -14385.576,E2 -14385.576} C_VEL
LIN {X 0,Y 333.828,Z 517.207,A -85,B 0,C 180,E1 -14389.077,E2 -14389.077} C_VEL
LIN {X 0,Y 334.018,Z 517.186,A -85,B 0,C 180,E1 -14392.747,E2 -14392.747} C_VEL
LIN {X 0,Y 333.807,Z 517.209,A -85,B 0,C 180,E1 -14395.168,E2 -14395.168} C_VEL
LIN {X 0,Y 334.123,Z 517.173,A -85,B 0,C 180,E1 -14397.588,E2 -14397.588} C_VEL
LIN {X 0,Y 334.257,Z 517.163,A -85,B 0,C 180,E1 -14399.999,E2 -14399.999} C_VEL
LIN {X 0,Y 334.098,Z 517.172,A -85,B 0,C 180,E1 -14402.411,E2 -14402.411} C_VEL
LIN {X 0,Y 334.014,Z 517.191,A -85,B 0,C 180,E1 -14407.252,E2 -14407.252} C_VEL
LIN {X 0,Y 333.827,Z 517.213,A -85,B 0,C 180,E1 -14410.922,E2 -14410.922} C_VEL
LIN {X 0,Y 333.797,Z 517.216,A -85,B 0,C 180,E1 -14414.634,E2 -14414.634} C_VEL
LIN {X 0,Y 333.787,Z 517.177,A -85,B 0,C 180,E1 -14418.656,E2 -14418.656} C_VEL
LIN {X 0,Y 333.723,Z 517.216,A -85,B 0,C 180,E1 -14422.275,E2 -14422.275} C_VEL
LIN {X 0,Y 333.727,Z 517.201,A -85,B 0,C 180,E1 -14426.246,E2 -14426.246} C_VEL
LIN {X 0,Y 333.701,Z 517.232,A -85,B 0,C 180,E1 -14428.972,E2 -14428.972} C_VEL
LIN {X 0,Y 333.662,Z 517.35,A -85,B 0,C 180,E1 -14432.342,E2 -14432.342} C_VEL
LIN {X 0,Y 335.32,Z 524.667,A -85,B 0,C 180,E1 -14435.933,E2 -14435.933} C_VEL
LIN {X 0,Y 337.046,Z 532.368,A -85,B 0,C 180,E1 -14439.513,E2 -14439.513} C_VEL
LIN {X 0,Y 338.899,Z 541.365,A -85,B 0,C 180,E1 -14443.465,E2 -14443.465} C_VEL
LIN {X 0,Y 340.281,Z 548.106,A -85,B 0,C 180,E1 -14446.292,E2 -14446.292} C_VEL
LIN {X 0,Y 340.893,Z 552.154,A -85,B 0,C 180,E1 -14447.918,E2 -14447.918} C_VEL
LIN {X 0,Y 340.264,Z 558.251,A -85,B 0,C 180,E1 -14450.189,E2 -14450.189} C_VEL
LIN {X 0,Y 339.791,Z 562.191,A -85,B 0,C 180,E1 -14451.555,E2 -14451.555} C_VEL
LIN {X 0,Y 340.95,Z 566.07,A -85,B 0,C 180,E1 -14451.842,E2 -14451.842} C_VEL
LIN {X 0,Y 346.409,Z 582.721,A -85,B 0,C 180,E1 -14453.14,E2 -14453.14} C_VEL
LIN {X 0,Y 349.263,Z 593.517,A -85,B 0,C 180,E1 -14453.961,E2 -14453.961} C_VEL
LIN {X 0,Y 352.555,Z 610.412,A -85,B 0,C 180,E1 -14455.292,E2 -14455.292} C_VEL
LIN {X 0,Y 354.795,Z 626.575,A -85,B 0,C 180,E1 -14456.685,E2 -14456.685} C_VEL
LIN {X 0,Y 355.455,Z 633.074,A -85,B 0,C 180,E1 -14457.281,E2 -14457.281} C_VEL
LIN {X 0,Y 353.104,Z 647.27,A -85,B 0,C 180,E1 -14458.337,E2 -14458.337} C_VEL
LIN {X 0,Y 350.239,Z 662.244,A -85,B 0,C 180,E1 -14459.708,E2 -14459.708} C_VEL
LIN {X 0,Y 347.374,Z 676.296,A -85,B 0,C 180,E1 -14461.283,E2 -14461.283} C_VEL
LIN {X 0,Y 344.633,Z 689.192,A -85,B 0,C 180,E1 -14463.018,E2 -14463.018} C_VEL
LIN {X 0,Y 341.842,Z 701.615,A -85,B 0,C 180,E1 -14464.999,E2 -14464.999} C_VEL
LIN {X 0,Y 339.294,Z 712.902,A -85,B 0,C 180,E1 -14467.148,E2 -14467.148} C_VEL
LIN {X 0,Y 337.287,Z 722.206,A -85,B 0,C 180,E1 -14469.256,E2 -14469.256} C_VEL
LIN {X 0,Y 335.54,Z 731.317,A -85,B 0,C 180,E1 -14471.69,E2 -14471.69} C_VEL
LIN {X 0,Y 334.073,Z 738.999,A -85,B 0,C 180,E1 -14474.13,E2 -14474.13} C_VEL
LIN {X 0,Y 333.193,Z 745.294,A -85,B 0,C 180,E1 -14476.585,E2 -14476.585} C_VEL
LIN {X 0,Y 332.505,Z 750.447,A -85,B 0,C 180,E1 -14479.035,E2 -14479.035} C_VEL
LIN {X 0,Y 332.238,Z 754.491,A -85,B 0,C 180,E1 -14481.486,E2 -14481.486} C_VEL
LIN {X 0,Y 332.217,Z 757.463,A -85,B 0,C 180,E1 -14483.93,E2 -14483.93} C_VEL
LIN {X 0,Y 332.137,Z 759.439,A -85,B 0,C 180,E1 -14486.362,E2 -14486.362} C_VEL
LIN {X 0,Y 332.343,Z 760.382,A -85,B 0,C 180,E1 -14488.79,E2 -14488.79} C_VEL
LIN {X 0,Y 332.346,Z 760.361,A -85,B 0,C 180,E1 -14491.213,E2 -14491.213} C_VEL
LIN {X 0,Y 332.142,Z 759.266,A -85,B 0,C 180,E1 -14493.641,E2 -14493.641} C_VEL
LIN {X 0,Y 332.282,Z 757.059,A -85,B 0,C 180,E1 -14496.24,E2 -14496.24} C_VEL
LIN {X 0,Y 332.264,Z 754.055,A -85,B 0,C 180,E1 -14498.516,E2 -14498.516} C_VEL
LIN {X 0,Y 332.529,Z 749.865,A -85,B 0,C 180,E1 -14500.967,E2 -14500.967} C_VEL
LIN {X 0,Y 333.199,Z 744.444,A -85,B 0,C 180,E1 -14503.417,E2 -14503.417} C_VEL
LIN {X 0,Y 334.08,Z 737.783,A -85,B 0,C 180,E1 -14505.873,E2 -14505.873} C_VEL
LIN {X 0,Y 335.466,Z 729.771,A -85,B 0,C 180,E1 -14508.317,E2 -14508.317} C_VEL
LIN {X 0,Y 337.19,Z 720.136,A -85,B 0,C 180,E1 -14510.753,E2 -14510.753} C_VEL
LIN {X 0,Y 339.443,Z 708.609,A -85,B 0,C 180,E1 -14513.166,E2 -14513.166} C_VEL
LIN {X 0,Y 341.848,Z 696.73,A -85,B 0,C 180,E1 -14515.233,E2 -14515.233} C_VEL
LIN {X 0,Y 344.301,Z 684.566,A -85,B 0,C 180,E1 -14517.013,E2 -14517.013} C_VEL
LIN {X 0,Y 346.71,Z 671.682,A -85,B 0,C 180,E1 -14518.614,E2 -14518.614} C_VEL
LIN {X 0,Y 351.366,Z 651.047,A -85,B 0,C 180,E1 -14521.002,E2 -14521.002} C_VEL
LIN {X 0,Y 355.146,Z 635.262,A -85,B 0,C 180,E1 -14522.543,E2 -14522.543} C_VEL
LIN {X 0,Y 355.608,Z 633.039,A -85,B 0,C 180,E1 -14522.741,E2 -14522.741} C_VEL
LIN {X 0,Y 355.551,Z 619.845,A -85,B 0,C 180,E1 -14524.288,E2 -14524.288} C_VEL
LIN {X 0,Y 356.029,Z 604.246,A -85,B 0,C 180,E1 -14525.97,E2 -14525.97} C_VEL
LIN {X 0,Y 355.462,Z 591.655,A -85,B 0,C 180,E1 -14527.504,E2 -14527.504} C_VEL
LIN {X 0,Y 354.486,Z 581.867,A -85,B 0,C 180,E1 -14528.908,E2 -14528.908} C_VEL
LIN {X 0,Y 353.668,Z 574.442,A -85,B 0,C 180,E1 -14530.131,E2 -14530.131} C_VEL
LIN {X 0,Y 352.626,Z 566.818,A -85,B 0,C 180,E1 -14531.665,E2 -14531.665} C_VEL
LIN {X 0,Y 352.097,Z 561.344,A -85,B 0,C 180,E1 -14532.995,E2 -14532.995} C_VEL
LIN {X 0,Y 351.587,Z 558.857,A -85,B 0,C 180,E1 -14533.978,E2 -14533.978} C_VEL
LIN {X 0,Y 351.232,Z 555.165,A -85,B 0,C 180,E1 -14536.084,E2 -14536.084} C_VEL
LIN {X 0,Y 351.83,Z 553.394,A -85,B 0,C 180,E1 -14537.655,E2 -14537.655} C_VEL
LIN {X 0,Y 352.774,Z 553.332,A -85,B 0,C 180,E1 -14539.205,E2 -14539.205} C_VEL
LIN {X 0,Y 354.395,Z 553.935,A -85,B 0,C 180,E1 -14540.662,E2 -14540.662} C_VEL
LIN {X 0,Y 356.91,Z 555.812,A -85,B 0,C 180,E1 -14542.38,E2 -14542.38} C_VEL
LIN {X 0,Y 360.097,Z 559.53,A -85,B 0,C 180,E1 -14544.162,E2 -14544.162} C_VEL
LIN {X 0,Y 362.856,Z 563.77,A -85,B 0,C 180,E1 -14545.539,E2 -14545.539} C_VEL
LIN {X 0,Y 363.895,Z 566.229,A -85,B 0,C 180,E1 -14546.148,E2 -14546.148} C_VEL
LIN {X 0,Y 364.325,Z 568.043,A -85,B 0,C 180,E1 -14546.478,E2 -14546.478} C_VEL
LIN {X 0,Y 360.402,Z 585.49,A -85,B 0,C 180,E1 -14548.074,E2 -14548.074} C_VEL
LIN {X 0,Y 356.496,Z 601.3,A -85,B 0,C 180,E1 -14549.821,E2 -14549.821} C_VEL
LIN {X 0,Y 352.412,Z 616.982,A -85,B 0,C 180,E1 -14551.915,E2 -14551.915} C_VEL
LIN {X 0,Y 348.809,Z 630.056,A -85,B 0,C 180,E1 -14554.009,E2 -14554.009} C_VEL
LIN {X 0,Y 345.421,Z 642.306,A -85,B 0,C 180,E1 -14556.377,E2 -14556.377} C_VEL
LIN {X 0,Y 342.567,Z 652.097,A -85,B 0,C 180,E1 -14558.645,E2 -14558.645} C_VEL
LIN {X 0,Y 340.424,Z 659.654,A -85,B 0,C 180,E1 -14560.712,E2 -14560.712} C_VEL
LIN {X 0,Y 338.394,Z 666.958,A -85,B 0,C 180,E1 -14563.097,E2 -14563.097} C_VEL
LIN {X 0,Y 336.67,Z 672.973,A -85,B 0,C 180,E1 -14565.493,E2 -14565.493} C_VEL
LIN {X 0,Y 335.4,Z 677.778,A -85,B 0,C 180,E1 -14567.905,E2 -14567.905} C_VEL
LIN {X 0,Y 334.479,Z 681.545,A -85,B 0,C 180,E1 -14570.323,E2 -14570.323} C_VEL
LIN {X 0,Y 333.822,Z 684.209,A -85,B 0,C 180,E1 -14572.744,E2 -14572.744} C_VEL
LIN {X 0,Y 333.314,Z 685.933,A -85,B 0,C 180,E1 -14575.162,E2 -14575.162} C_VEL
LIN {X 0,Y 332.865,Z 686.698,A -85,B 0,C 180,E1 -14577.58,E2 -14577.58} C_VEL
LIN {X 0,Y 332.662,Z 686.44,A -85,B 0,C 180,E1 -14580.001,E2 -14580.001} C_VEL
LIN {X 0,Y 332.826,Z 685.245,A -85,B 0,C 180,E1 -14582.421,E2 -14582.421} C_VEL
LIN {X 0,Y 333.008,Z 682.988,A -85,B 0,C 180,E1 -14584.843,E2 -14584.843} C_VEL
LIN {X 0,Y 333.298,Z 679.131,A -85,B 0,C 180,E1 -14587.665,E2 -14587.665} C_VEL
LIN {X 0,Y 333.74,Z 674.203,A -85,B 0,C 180,E1 -14590.312,E2 -14590.312} C_VEL
LIN {X 0,Y 334.393,Z 668.444,A -85,B 0,C 180,E1 -14592.75,E2 -14592.75} C_VEL
LIN {X 0,Y 335.548,Z 660.828,A -85,B 0,C 180,E1 -14595.351,E2 -14595.351} C_VEL
LIN {X 0,Y 336.989,Z 651.688,A -85,B 0,C 180,E1 -14597.916,E2 -14597.916} C_VEL
LIN {X 0,Y 338.782,Z 641.311,A -85,B 0,C 180,E1 -14600.334,E2 -14600.334} C_VEL
LIN {X 0,Y 340.552,Z 630.623,A -85,B 0,C 180,E1 -14602.445,E2 -14602.445} C_VEL
LIN {X 0,Y 342.792,Z 618.107,A -85,B 0,C 180,E1 -14604.531,E2 -14604.531} C_VEL
LIN {X 0,Y 345.108,Z 604.491,A -85,B 0,C 180,E1 -14606.446,E2 -14606.446} C_VEL
LIN {X 0,Y 347.501,Z 589.473,A -85,B 0,C 180,E1 -14608.213,E2 -14608.213} C_VEL
LIN {X 0,Y 349.731,Z 574.674,A -85,B 0,C 180,E1 -14609.66,E2 -14609.66} C_VEL
LIN {X 0,Y 351.472,Z 559.585,A -85,B 0,C 180,E1 -14610.905,E2 -14610.905} C_VEL
LIN {X 0,Y 345.504,Z 544.333,A -85,B 0,C 180,E1 -14612.571,E2 -14612.571} C_VEL
LIN {X 0,Y 338.336,Z 527.856,A -85,B 0,C 180,E1 -14614.258,E2 -14614.258} C_VEL
LIN {X 0,Y 333.799,Z 517.935,A -85,B 0,C 180,E1 -14615.21,E2 -14615.21} C_VEL
LIN {X 0,Y 333.689,Z 517.232,A -85,B 0,C 180,E1 -14615.259,E2 -14615.259} C_VEL
LIN {X 0,Y 333.653,Z 517.238,A -85,B 0,C 180,E1 -14619.192,E2 -14619.192} C_VEL
LIN {X 0,Y 333.638,Z 517.239,A -85,B 0,C 180,E1 -14622.5,E2 -14622.5} C_VEL
LIN {X 0,Y 333.602,Z 517.245,A -85,B 0,C 180,E1 -14625.955,E2 -14625.955} C_VEL
LIN {X 0,Y 333.653,Z 517.237,A -85,B 0,C 180,E1 -14629.315,E2 -14629.315} C_VEL
LIN {X 0,Y 333.671,Z 517.233,A -85,B 0,C 180,E1 -14633.167,E2 -14633.167} C_VEL
LIN {X 0,Y 333.68,Z 517.234,A -85,B 0,C 180,E1 -14635.341,E2 -14635.341} C_VEL
LIN {X 0,Y 333.693,Z 517.373,A -85,B 0,C 180,E1 -14638.494,E2 -14638.494} C_VEL
LIN {X 0,Y 334.689,Z 522.355,A -85,B 0,C 180,E1 -14641.879,E2 -14641.879} C_VEL
LIN {X 0,Y 335.124,Z 526.165,A -85,B 0,C 180,E1 -14644.393,E2 -14644.393} C_VEL
LIN {X 0,Y 335.201,Z 530.634,A -85,B 0,C 180,E1 -14647.3,E2 -14647.3} C_VEL
LIN {X 0,Y 335.189,Z 532.163,A -85,B 0,C 180,E1 -14648.281,E2 -14648.281} C_VEL
LIN {X 0,Y 336.495,Z 535.509,A -85,B 0,C 180,E1 -14648.512,E2 -14648.512} C_VEL
LIN {X 0,Y 344.066,Z 552.82,A -85,B 0,C 180,E1 -14649.864,E2 -14649.864} C_VEL
LIN {X 0,Y 349.285,Z 566.914,A -85,B 0,C 180,E1 -14651.032,E2 -14651.032} C_VEL
LIN {X 0,Y 353.961,Z 581.72,A -85,B 0,C 180,E1 -14652.376,E2 -14652.376} C_VEL
LIN {X 0,Y 355.008,Z 585.459,A -85,B 0,C 180,E1 -14652.724,E2 -14652.724} C_VEL
LIN {X 0,Y 353.061,Z 601.44,A -85,B 0,C 180,E1 -14653.817,E2 -14653.817} C_VEL
LIN {X 0,Y 350.898,Z 615.969,A -85,B 0,C 180,E1 -14655.055,E2 -14655.055} C_VEL
LIN {X 0,Y 348.665,Z 629.468,A -85,B 0,C 180,E1 -14656.447,E2 -14656.447} C_VEL
LIN {X 0,Y 346.032,Z 643.192,A -85,B 0,C 180,E1 -14658.132,E2 -14658.132} C_VEL
LIN {X 0,Y 343.66,Z 655.72,A -85,B 0,C 180,E1 -14659.988,E2 -14659.988} C_VEL
LIN {X 0,Y 341.239,Z 667.216,A -85,B 0,C 180,E1 -14662.008,E2 -14662.008} C_VEL
LIN {X 0,Y 338.894,Z 678.289,A -85,B 0,C 180,E1 -14664.346,E2 -14664.346} C_VEL
LIN {X 0,Y 337.126,Z 686.515,A -85,B 0,C 180,E1 -14666.413,E2 -14666.413} C_VEL
LIN {X 0,Y 335.555,Z 694.534,A -85,B 0,C 180,E1 -14668.799,E2 -14668.799} C_VEL
LIN {X 0,Y 334.284,Z 701.193,A -85,B 0,C 180,E1 -14671.203,E2 -14671.203} C_VEL
LIN {X 0,Y 333.408,Z 706.621,A -85,B 0,C 180,E1 -14673.624,E2 -14673.624} C_VEL
LIN {X 0,Y 332.807,Z 711.016,A -85,B 0,C 180,E1 -14676.06,E2 -14676.06} C_VEL
LIN {X 0,Y 332.355,Z 714.297,A -85,B 0,C 180,E1 -14678.511,E2 -14678.511} C_VEL
LIN {X 0,Y 332.079,Z 716.638,A -85,B 0,C 180,E1 -14680.979,E2 -14680.979} C_VEL
LIN {X 0,Y 331.987,Z 717.965,A -85,B 0,C 180,E1 -14683.464,E2 -14683.464} C_VEL
LIN {X 0,Y 331.909,Z 718.331,A -85,B 0,C 180,E1 -14685.976,E2 -14685.976} C_VEL
LIN {X 0,Y 332.048,Z 717.71,A -85,B 0,C 180,E1 -14688.509,E2 -14688.509} C_VEL
LIN {X 0,Y 332.411,Z 715.62,A -85,B 0,C 180,E1 -14691.521,E2 -14691.521} C_VEL
LIN {X 0,Y 332.832,Z 713.298,A -85,B 0,C 180,E1 -14693.651,E2 -14693.651} C_VEL
LIN {X 0,Y 333.648,Z 709.363,A -85,B 0,C 180,E1 -14696.252,E2 -14696.252} C_VEL
LIN {X 0,Y 334.698,Z 704.189,A -85,B 0,C 180,E1 -14698.877,E2 -14698.877} C_VEL
LIN {X 0,Y 336.163,Z 697.667,A -85,B 0,C 180,E1 -14701.509,E2 -14701.509} C_VEL
LIN {X 0,Y 338.176,Z 689.606,A -85,B 0,C 180,E1 -14704.131,E2 -14704.131} C_VEL
LIN {X 0,Y 340.282,Z 681.348,A -85,B 0,C 180,E1 -14706.342,E2 -14706.342} C_VEL
LIN {X 0,Y 342.79,Z 671.611,A -85,B 0,C 180,E1 -14708.536,E2 -14708.536} C_VEL
LIN {X 0,Y 345.52,Z 660.717,A -85,B 0,C 180,E1 -14710.607,E2 -14710.607} C_VEL
LIN {X 0,Y 346.557,Z 656.521,A -85,B 0,C 180,E1 -14711.318,E2 -14711.318} C_VEL
LIN {X 0,Y 347.049,Z 652.502,A -85,B 0,C 180,E1 -14712.029,E2 -14712.029} C_VEL
LIN {X 0,Y 346.215,Z 646.035,A -85,B 0,C 180,E1 -14713.266,E2 -14713.266} C_VEL
LIN {X 0,Y 345.352,Z 639.224,A -85,B 0,C 180,E1 -14714.45,E2 -14714.45} C_VEL
LIN {X 0,Y 345.769,Z 634.67,A -85,B 0,C 180,E1 -14715.068,E2 -14715.068} C_VEL
LIN {X 0,Y 348.763,Z 620.539,A -85,B 0,C 180,E1 -14716.614,E2 -14716.614} C_VEL
LIN {X 0,Y 351.349,Z 606.17,A -85,B 0,C 180,E1 -14717.91,E2 -14717.91} C_VEL
LIN {X 0,Y 353.824,Z 590.51,A -85,B 0,C 180,E1 -14719.043,E2 -14719.043} C_VEL
LIN {X 0,Y 349.797,Z 576.656,A -85,B 0,C 180,E1 -14720.643,E2 -14720.643} C_VEL
LIN {X 0,Y 345.269,Z 564.706,A -85,B 0,C 180,E1 -14722.027,E2 -14722.027} C_VEL
LIN {X 0,Y 338.617,Z 550.565,A -85,B 0,C 180,E1 -14723.732,E2 -14723.732} C_VEL
LIN {X 0,Y 334.178,Z 542.519,A -85,B 0,C 180,E1 -14724.751,E2 -14724.751} C_VEL
LIN {X 0,Y 331.834,Z 538.559,A -85,B 0,C 180,E1 -14725.273,E2 -14725.273} C_VEL
LIN {X 0,Y 330.063,Z 535.664,A -85,B 0,C 180,E1 -14725.671,E2 -14725.671} C_VEL
LIN {X 0,Y 329.615,Z 534.359,A -85,B 0,C 180,E1 -14725.835,E2 -14725.835} C_VEL
LIN {X 0,Y 329.095,Z 529.999,A -85,B 0,C 180,E1 -14729.167,E2 -14729.167} C_VEL
LIN {X 0,Y 328.465,Z 526.543,A -85,B 0,C 180,E1 -14731.918,E2 -14731.918} C_VEL
LIN {X 0,Y 327.842,Z 523.183,A -85,B 0,C 180,E1 -14734.612,E2 -14734.612} C_VEL
LIN {X 0,Y 326.656,Z 518.12,A -85,B 0,C 180,E1 -14738.835,E2 -14738.835} C_VEL
LIN {X 0,Y 326.735,Z 518.094,A -85,B 0,C 180,E1 -14741.176,E2 -14741.176} C_VEL
LIN {X 0,Y 326.754,Z 518.093,A -85,B 0,C 180,E1 -14745.432,E2 -14745.432} C_VEL
LIN {X 0,Y 326.764,Z 518.087,A -85,B 0,C 180,E1 -14748.838,E2 -14748.838} C_VEL
LIN {X 0,Y 326.971,Z 518.062,A -85,B 0,C 180,E1 -14752.59,E2 -14752.59} C_VEL
LIN {X 0,Y 326.774,Z 518.085,A -85,B 0,C 180,E1 -14755.064,E2 -14755.064} C_VEL
LIN {X 0,Y 327.06,Z 518.053,A -85,B 0,C 180,E1 -14757.536,E2 -14757.536} C_VEL
LIN {X 0,Y 327.208,Z 518.041,A -85,B 0,C 180,E1 -14759.999,E2 -14759.999} C_VEL
LIN {X 0,Y 327.039,Z 518.052,A -85,B 0,C 180,E1 -14762.463,E2 -14762.463} C_VEL
LIN {X 0,Y 326.986,Z 518.057,A -85,B 0,C 180,E1 -14766.169,E2 -14766.169} C_VEL
LIN {X 0,Y 326.904,Z 518.065,A -85,B 0,C 180,E1 -14768.655,E2 -14768.655} C_VEL
LIN {X 0,Y 326.728,Z 518.086,A -85,B 0,C 180,E1 -14772.421,E2 -14772.421} C_VEL
LIN {X 0,Y 326.743,Z 518.09,A -85,B 0,C 180,E1 -14774.957,E2 -14774.957} C_VEL
LIN {X 0,Y 326.753,Z 518.055,A -85,B 0,C 180,E1 -14778.854,E2 -14778.854} C_VEL
LIN {X 0,Y 326.677,Z 518.08,A -85,B 0,C 180,E1 -14782.783,E2 -14782.783} C_VEL
LIN {X 0,Y 326.676,Z 518.093,A -85,B 0,C 180,E1 -14786.858,E2 -14786.858} C_VEL
LIN {X 0,Y 326.629,Z 518.112,A -85,B 0,C 180,E1 -14790.612,E2 -14790.612} C_VEL
LIN {X 0,Y 326.585,Z 518.12,A -85,B 0,C 180,E1 -14791.637,E2 -14791.637} C_VEL
LIN {X 0,Y 328.373,Z 525.986,A -85,B 0,C 180,E1 -14795.584,E2 -14795.584} C_VEL
LIN {X 0,Y 330.275,Z 534.63,A -85,B 0,C 180,E1 -14799.67,E2 -14799.67} C_VEL
LIN {X 0,Y 331.997,Z 542.9,A -85,B 0,C 180,E1 -14803.354,E2 -14803.354} C_VEL
LIN {X 0,Y 333.552,Z 550.607,A -85,B 0,C 180,E1 -14806.627,E2 -14806.627} C_VEL
LIN {X 0,Y 333.946,Z 554.184,A -85,B 0,C 180,E1 -14808.075,E2 -14808.075} C_VEL
LIN {X 0,Y 333.19,Z 560.49,A -85,B 0,C 180,E1 -14810.452,E2 -14810.452} C_VEL
LIN {X 0,Y 334.304,Z 564.493,A -85,B 0,C 180,E1 -14810.756,E2 -14810.756} C_VEL
LIN {X 0,Y 335.154,Z 566.806,A -85,B 0,C 180,E1 -14810.961,E2 -14810.961} C_VEL
LIN {X 0,Y 340.922,Z 584.505,A -85,B 0,C 180,E1 -14812.407,E2 -14812.407} C_VEL
LIN {X 0,Y 343.956,Z 596.924,A -85,B 0,C 180,E1 -14813.405,E2 -14813.405} C_VEL
LIN {X 0,Y 346.953,Z 613.337,A -85,B 0,C 180,E1 -14814.766,E2 -14814.766} C_VEL
LIN {X 0,Y 348.969,Z 629.818,A -85,B 0,C 180,E1 -14816.26,E2 -14816.26} C_VEL
LIN {X 0,Y 349.404,Z 633.723,A -85,B 0,C 180,E1 -14816.653,E2 -14816.653} C_VEL
LIN {X 0,Y 347.097,Z 647.64,A -85,B 0,C 180,E1 -14817.723,E2 -14817.723} C_VEL
LIN {X 0,Y 344.057,Z 662.813,A -85,B 0,C 180,E1 -14819.148,E2 -14819.148} C_VEL
LIN {X 0,Y 341.124,Z 676.388,A -85,B 0,C 180,E1 -14820.707,E2 -14820.707} C_VEL
LIN {X 0,Y 338.265,Z 689.179,A -85,B 0,C 180,E1 -14822.467,E2 -14822.467} C_VEL
LIN {X 0,Y 335.45,Z 701.109,A -85,B 0,C 180,E1 -14824.408,E2 -14824.408} C_VEL
LIN {X 0,Y 332.677,Z 712.742,A -85,B 0,C 180,E1 -14826.667,E2 -14826.667} C_VEL
LIN {X 0,Y 330.312,Z 723.035,A -85,B 0,C 180,E1 -14829.07,E2 -14829.07} C_VEL
LIN {X 0,Y 328.483,Z 732.079,A -85,B 0,C 180,E1 -14831.606,E2 -14831.606} C_VEL
LIN {X 0,Y 326.852,Z 740.336,A -85,B 0,C 180,E1 -14834.41,E2 -14834.41} C_VEL
LIN {X 0,Y 325.982,Z 746.372,A -85,B 0,C 180,E1 -14836.918,E2 -14836.918} C_VEL
LIN {X 0,Y 325.294,Z 752.254,A -85,B 0,C 180,E1 -14840.048,E2 -14840.048} C_VEL
LIN {X 0,Y 325.15,Z 755.7,A -85,B 0,C 180,E1 -14842.55,E2 -14842.55} C_VEL
LIN {X 0,Y 325.069,Z 758.173,A -85,B 0,C 180,E1 -14845.04,E2 -14845.04} C_VEL
LIN {X 0,Y 325.105,Z 759.586,A -85,B 0,C 180,E1 -14847.523,E2 -14847.523} C_VEL
LIN {X 0,Y 325.257,Z 760.052,A -85,B 0,C 180,E1 -14850.001,E2 -14850.001} C_VEL
LIN {X 0,Y 325.284,Z 759.905,A -85,B 0,C 180,E1 -14851.239,E2 -14851.239} C_VEL
LIN {X 0,Y 325.068,Z 758.784,A -85,B 0,C 180,E1 -14853.72,E2 -14853.72} C_VEL
LIN {X 0,Y 325.19,Z 756.737,A -85,B 0,C 180,E1 -14856.205,E2 -14856.205} C_VEL
LIN {X 0,Y 325.202,Z 753.528,A -85,B 0,C 180,E1 -14858.702,E2 -14858.702} C_VEL
LIN {X 0,Y 325.495,Z 749.304,A -85,B 0,C 180,E1 -14861.207,E2 -14861.207} C_VEL
LIN {X 0,Y 326.193,Z 743.865,A -85,B 0,C 180,E1 -14863.711,E2 -14863.711} C_VEL
LIN {X 0,Y 327.121,Z 737.169,A -85,B 0,C 180,E1 -14866.219,E2 -14866.219} C_VEL
LIN {X 0,Y 328.587,Z 729.118,A -85,B 0,C 180,E1 -14868.714,E2 -14868.714} C_VEL
LIN {X 0,Y 330.422,Z 719.449,A -85,B 0,C 180,E1 -14871.199,E2 -14871.199} C_VEL
LIN {X 0,Y 332.805,Z 707.865,A -85,B 0,C 180,E1 -14873.656,E2 -14873.656} C_VEL
LIN {X 0,Y 335.068,Z 696.949,A -85,B 0,C 180,E1 -14875.59,E2 -14875.59} C_VEL
LIN {X 0,Y 337.63,Z 684.758,A -85,B 0,C 180,E1 -14877.423,E2 -14877.423} C_VEL
LIN {X 0,Y 340.72,Z 670.32,A -85,B 0,C 180,E1 -14879.334,E2 -14879.334} C_VEL
LIN {X 0,Y 344.137,Z 656.783,A -85,B 0,C 180,E1 -14881.043,E2 -14881.043} C_VEL
LIN {X 0,Y 348.033,Z 641.5,A -85,B 0,C 180,E1 -14882.697,E2 -14882.697} C_VEL
LIN {X 0,Y 349.736,Z 634.469,A -85,B 0,C 180,E1 -14883.389,E2 -14883.389} C_VEL
LIN {X 0,Y 350.145,Z 620.664,A -85,B 0,C 180,E1 -14885.069,E2 -14885.069} C_VEL
LIN {X 0,Y 350.965,Z 605.862,A -85,B 0,C 180,E1 -14886.776,E2 -14886.776} C_VEL
LIN {X 0,Y 350.791,Z 594.432,A -85,B 0,C 180,E1 -14888.276,E2 -14888.276} C_VEL
LIN {X 0,Y 350.296,Z 585.936,A -85,B 0,C 180,E1 -14889.562,E2 -14889.562} C_VEL
LIN {X 0,Y 349.759,Z 578.47,A -85,B 0,C 180,E1 -14890.874,E2 -14890.874} C_VEL
LIN {X 0,Y 349.269,Z 571.722,A -85,B 0,C 180,E1 -14892.313,E2 -14892.313} C_VEL
LIN {X 0,Y 349.066,Z 566.884,A -85,B 0,C 180,E1 -14893.547,E2 -14893.547} C_VEL
LIN {X 0,Y 348.594,Z 563.508,A -85,B 0,C 180,E1 -14895.12,E2 -14895.12} C_VEL
LIN {X 0,Y 348.791,Z 561.114,A -85,B 0,C 180,E1 -14896.758,E2 -14896.758} C_VEL
LIN {X 0,Y 349.462,Z 559.932,A -85,B 0,C 180,E1 -14898.083,E2 -14898.083} C_VEL
LIN {X 0,Y 351.013,Z 560.259,A -85,B 0,C 180,E1 -14900.156,E2 -14900.156} C_VEL
LIN {X 0,Y 353.358,Z 561.73,A -85,B 0,C 180,E1 -14901.935,E2 -14901.935} C_VEL
LIN {X 0,Y 355.36,Z 563.94,A -85,B 0,C 180,E1 -14903.263,E2 -14903.263} C_VEL
LIN {X 0,Y 357.691,Z 567.328,A -85,B 0,C 180,E1 -14904.616,E2 -14904.616} C_VEL
LIN {X 0,Y 359.497,Z 570.976,A -85,B 0,C 180,E1 -14905.687,E2 -14905.687} C_VEL
LIN {X 0,Y 359.548,Z 571.924,A -85,B 0,C 180,E1 -14905.843,E2 -14905.843} C_VEL
LIN {X 0,Y 355,Z 589.507,A -85,B 0,C 180,E1 -14907.521,E2 -14907.521} C_VEL
LIN {X 0,Y 350.908,Z 604.662,A -85,B 0,C 180,E1 -14909.29,E2 -14909.29} C_VEL
LIN {X 0,Y 346.893,Z 618.708,A -85,B 0,C 180,E1 -14911.239,E2 -14911.239} C_VEL
LIN {X 0,Y 343.274,Z 630.832,A -85,B 0,C 180,E1 -14913.23,E2 -14913.23} C_VEL
LIN {X 0,Y 339.72,Z 642.688,A -85,B 0,C 180,E1 -14915.56,E2 -14915.56} C_VEL
LIN {X 0,Y 336.588,Z 652.766,A -85,B 0,C 180,E1 -14917.924,E2 -14917.924} C_VEL
LIN {X 0,Y 333.927,Z 661.271,A -85,B 0,C 180,E1 -14920.322,E2 -14920.322} C_VEL
LIN {X 0,Y 331.763,Z 668.441,A -85,B 0,C 180,E1 -14922.749,E2 -14922.749} C_VEL
LIN {X 0,Y 329.92,Z 674.353,A -85,B 0,C 180,E1 -14925.19,E2 -14925.19} C_VEL
LIN {X 0,Y 328.568,Z 679.035,A -85,B 0,C 180,E1 -14927.65,E2 -14927.65} C_VEL
LIN {X 0,Y 327.554,Z 682.691,A -85,B 0,C 180,E1 -14930.117,E2 -14930.117} C_VEL
LIN {X 0,Y 326.867,Z 685.296,A -85,B 0,C 180,E1 -14932.588,E2 -14932.588} C_VEL
LIN {X 0,Y 326.307,Z 686.909,A -85,B 0,C 180,E1 -14935.058,E2 -14935.058} C_VEL
LIN {X 0,Y 325.831,Z 687.621,A -85,B 0,C 180,E1 -14937.528,E2 -14937.528} C_VEL
LIN {X 0,Y 325.616,Z 687.28,A -85,B 0,C 180,E1 -14940.001,E2 -14940.001} C_VEL
LIN {X 0,Y 325.792,Z 685.996,A -85,B 0,C 180,E1 -14942.473,E2 -14942.473} C_VEL
LIN {X 0,Y 325.978,Z 684.949,A -85,B 0,C 180,E1 -14943.709,E2 -14943.709} C_VEL
LIN {X 0,Y 325.97,Z 682.147,A -85,B 0,C 180,E1 -14946.189,E2 -14946.189} C_VEL
LIN {X 0,Y 326.387,Z 678.331,A -85,B 0,C 180,E1 -14948.67,E2 -14948.67} C_VEL
LIN {X 0,Y 326.874,Z 673.325,A -85,B 0,C 180,E1 -14951.158,E2 -14951.158} C_VEL
LIN {X 0,Y 327.684,Z 667.142,A -85,B 0,C 180,E1 -14953.647,E2 -14953.647} C_VEL
LIN {X 0,Y 328.895,Z 659.647,A -85,B 0,C 180,E1 -14956.129,E2 -14956.129} C_VEL
LIN {X 0,Y 330.396,Z 650.65,A -85,B 0,C 180,E1 -14958.607,E2 -14958.607} C_VEL
LIN {X 0,Y 332.293,Z 639.894,A -85,B 0,C 180,E1 -14961.073,E2 -14961.073} C_VEL
LIN {X 0,Y 334.198,Z 628.783,A -85,B 0,C 180,E1 -14963.223,E2 -14963.223} C_VEL
LIN {X 0,Y 336.563,Z 615.774,A -85,B 0,C 180,E1 -14965.346,E2 -14965.346} C_VEL
LIN {X 0,Y 338.837,Z 602.697,A -85,B 0,C 180,E1 -14967.15,E2 -14967.15} C_VEL
LIN {X 0,Y 341.064,Z 588.673,A -85,B 0,C 180,E1 -14968.795,E2 -14968.795} C_VEL
LIN {X 0,Y 343.485,Z 573.653,A -85,B 0,C 180,E1 -14970.256,E2 -14970.256} C_VEL
LIN {X 0,Y 344.972,Z 561.853,A -85,B 0,C 180,E1 -14971.237,E2 -14971.237} C_VEL
LIN {X 0,Y 339.169,Z 546.932,A -85,B 0,C 180,E1 -14972.942,E2 -14972.942} C_VEL
LIN {X 0,Y 332.459,Z 531.291,A -85,B 0,C 180,E1 -14974.614,E2 -14974.614} C_VEL
LIN {X 0,Y 326.743,Z 518.688,A -85,B 0,C 180,E1 -14975.851,E2 -14975.851} C_VEL
LIN {X 0,Y 326.642,Z 518.112,A -85,B 0,C 180,E1 -14975.895,E2 -14975.895} C_VEL
LIN {X 0,Y 326.618,Z 518.114,A -85,B 0,C 180,E1 -14979.227,E2 -14979.227} C_VEL
LIN {X 0,Y 326.581,Z 518.119,A -85,B 0,C 180,E1 -14982.972,E2 -14982.972} C_VEL
LIN {X 0,Y 326.582,Z 518.117,A -85,B 0,C 180,E1 -14987.028,E2 -14987.028} C_VEL
LIN {X 0,Y 326.617,Z 518.114,A -85,B 0,C 180,E1 -14990.773,E2 -14990.773} C_VEL
LIN {X 0,Y 326.619,Z 518.117,A -85,B 0,C 180,E1 -14994.48,E2 -14994.48} C_VEL
LIN {X 0,Y 326.611,Z 518.168,A -85,B 0,C 180,E1 -14997.82,E2 -14997.82} C_VEL
LIN {X 0,Y 327.391,Z 521.954,A -85,B 0,C 180,E1 -15000.413,E2 -15000.413} C_VEL
LIN {X 0,Y 328.075,Z 526.113,A -85,B 0,C 180,E1 -15003.264,E2 -15003.264} C_VEL
LIN {X 0,Y 328.322,Z 530.259,A -85,B 0,C 180,E1 -15006.001,E2 -15006.001} C_VEL
LIN {X 0,Y 328.271,Z 532.545,A -85,B 0,C 180,E1 -15007.488,E2 -15007.488} C_VEL
LIN {X 0,Y 329.579,Z 535.827,A -85,B 0,C 180,E1 -15007.738,E2 -15007.738} C_VEL
LIN {X 0,Y 337.033,Z 552.571,A -85,B 0,C 180,E1 -15009.102,E2 -15009.102} C_VEL
LIN {X 0,Y 343.003,Z 568.587,A -85,B 0,C 180,E1 -15010.481,E2 -15010.481} C_VEL
LIN {X 0,Y 347.8,Z 584.057,A -85,B 0,C 180,E1 -15011.937,E2 -15011.937} C_VEL
LIN {X 0,Y 348.687,Z 587.404,A -85,B 0,C 180,E1 -15012.268,E2 -15012.268} C_VEL
LIN {X 0,Y 346.737,Z 602.466,A -85,B 0,C 180,E1 -15013.321,E2 -15013.321} C_VEL
LIN {X 0,Y 344.417,Z 617.326,A -85,B 0,C 180,E1 -15014.616,E2 -15014.616} C_VEL
LIN {X 0,Y 342.125,Z 630.667,A -85,B 0,C 180,E1 -15016.031,E2 -15016.031} C_VEL
LIN {X 0,Y 339.4,Z 644.28,A -85,B 0,C 180,E1 -15017.745,E2 -15017.745} C_VEL
LIN {X 0,Y 337.129,Z 655.857,A -85,B 0,C 180,E1 -15019.489,E2 -15019.489} C_VEL
LIN {X 0,Y 334.645,Z 667.381,A -85,B 0,C 180,E1 -15021.545,E2 -15021.545} C_VEL
LIN {X 0,Y 332.184,Z 678.505,A -85,B 0,C 180,E1 -15023.926,E2 -15023.926} C_VEL
LIN {X 0,Y 330.092,Z 687.856,A -85,B 0,C 180,E1 -15026.337,E2 -15026.337} C_VEL
LIN {X 0,Y 328.481,Z 695.708,A -85,B 0,C 180,E1 -15028.773,E2 -15028.773} C_VEL
LIN {X 0,Y 327.202,Z 702.283,A -85,B 0,C 180,E1 -15031.229,E2 -15031.229} C_VEL
LIN {X 0,Y 326.165,Z 708.773,A -85,B 0,C 180,E1 -15034.324,E2 -15034.324} C_VEL
LIN {X 0,Y 325.46,Z 713.596,A -85,B 0,C 180,E1 -15037.443,E2 -15037.443} C_VEL
LIN {X 0,Y 325.096,Z 716.265,A -85,B 0,C 180,E1 -15039.958,E2 -15039.958} C_VEL
LIN {X 0,Y 324.957,Z 718.022,A -85,B 0,C 180,E1 -15042.489,E2 -15042.489} C_VEL
LIN {X 0,Y 324.855,Z 718.752,A -85,B 0,C 180,E1 -15045.045,E2 -15045.045} C_VEL
LIN {X 0,Y 324.978,Z 718.422,A -85,B 0,C 180,E1 -15047.907,E2 -15047.907} C_VEL
LIN {X 0,Y 325.115,Z 717.279,A -85,B 0,C 180,E1 -15050.233,E2 -15050.233} C_VEL
LIN {X 0,Y 325.575,Z 714.941,A -85,B 0,C 180,E1 -15052.863,E2 -15052.863} C_VEL
LIN {X 0,Y 326.311,Z 711.537,A -85,B 0,C 180,E1 -15055.514,E2 -15055.514} C_VEL
LIN {X 0,Y 327.433,Z 706.537,A -85,B 0,C 180,E1 -15058.354,E2 -15058.354} C_VEL
LIN {X 0,Y 328.988,Z 699.818,A -85,B 0,C 180,E1 -15061.294,E2 -15061.294} C_VEL
LIN {X 0,Y 330.641,Z 693.438,A -85,B 0,C 180,E1 -15063.547,E2 -15063.547} C_VEL
LIN {X 0,Y 332.748,Z 685.605,A -85,B 0,C 180,E1 -15065.879,E2 -15065.879} C_VEL
LIN {X 0,Y 335.307,Z 676.207,A -85,B 0,C 180,E1 -15068.191,E2 -15068.191} C_VEL
LIN {X 0,Y 337.859,Z 666.776,A -85,B 0,C 180,E1 -15070.152,E2 -15070.152} C_VEL
LIN {X 0,Y 340.548,Z 656.369,A -85,B 0,C 180,E1 -15072.016,E2 -15072.016} C_VEL
LIN {X 0,Y 343.557,Z 644.048,A -85,B 0,C 180,E1 -15073.863,E2 -15073.863} C_VEL
LIN {X 0,Y 345.769,Z 634.67,A -85,B 0,C 180,E1 -15075.068,E2 -15075.068} C_VEL
LIN {X 0,Y 346.21,Z 630.081,A -85,B 0,C 180,E1 -15075.671,E2 -15075.671} C_VEL
LIN {X 0,Y 344.681,Z 615.043,A -85,B 0,C 180,E1 -15077.809,E2 -15077.809} C_VEL
LIN {X 0,Y 345.048,Z 610.043,A -85,B 0,C 180,E1 -15078.325,E2 -15078.325} C_VEL
LIN {X 0,Y 347.654,Z 595.016,A -85,B 0,C 180,E1 -15079.492,E2 -15079.492} C_VEL
LIN {X 0,Y 347.846,Z 592.076,A -85,B 0,C 180,E1 -15079.718,E2 -15079.718} C_VEL
LIN {X 0,Y 344.127,Z 579.178,A -85,B 0,C 180,E1 -15081.284,E2 -15081.284} C_VEL
LIN {X 0,Y 339.41,Z 566.573,A -85,B 0,C 180,E1 -15082.816,E2 -15082.816} C_VEL
LIN {X 0,Y 332.991,Z 552.765,A -85,B 0,C 180,E1 -15084.572,E2 -15084.572} C_VEL
LIN {X 0,Y 327.614,Z 543.264,A -85,B 0,C 180,E1 -15085.867,E2 -15085.867} C_VEL
LIN {X 0,Y 325.19,Z 539.293,A -85,B 0,C 180,E1 -15086.433,E2 -15086.433} C_VEL
LIN {X 0,Y 323.083,Z 536.07,A -85,B 0,C 180,E1 -15086.931,E2 -15086.931} C_VEL
LIN {X 0,Y 322.672,Z 534.887,A -85,B 0,C 180,E1 -15087.099,E2 -15087.099} C_VEL
LIN {X 0,Y 321.969,Z 530.202,A -85,B 0,C 180,E1 -15090.82,E2 -15090.82} C_VEL
LIN {X 0,Y 321.296,Z 526.247,A -85,B 0,C 180,E1 -15094.056,E2 -15094.056} C_VEL
LIN {X 0,Y 320.208,Z 521.524,A -85,B 0,C 180,E1 -15098.091,E2 -15098.091} C_VEL
LIN {X 0,Y 319.625,Z 518.983,A -85,B 0,C 180,E1 -15100.407,E2 -15100.407} C_VEL
LIN {X 0,Y 319.664,Z 518.973,A -85,B 0,C 180,E1 -15103.392,E2 -15103.392} C_VEL
LIN {X 0,Y 319.723,Z 518.965,A -85,B 0,C 180,E1 -15106.007,E2 -15106.007} C_VEL
LIN {X 0,Y 319.75,Z 518.965,A -85,B 0,C 180,E1 -15109.872,E2 -15109.872} C_VEL
LIN {X 0,Y 319.925,Z 518.939,A -85,B 0,C 180,E1 -15112.425,E2 -15112.425} C_VEL
LIN {X 0,Y 319.743,Z 518.96,A -85,B 0,C 180,E1 -15114.955,E2 -15114.955} C_VEL
LIN {X 0,Y 320,Z 518.933,A -85,B 0,C 180,E1 -15117.482,E2 -15117.482} C_VEL
LIN {X 0,Y 320.159,Z 518.919,A -85,B 0,C 180,E1 -15119.999,E2 -15119.999} C_VEL
LIN {X 0,Y 319.982,Z 518.93,A -85,B 0,C 180,E1 -15122.517,E2 -15122.517} C_VEL
LIN {X 0,Y 319.941,Z 518.935,A -85,B 0,C 180,E1 -15126.305,E2 -15126.305} C_VEL
LIN {X 0,Y 319.832,Z 518.945,A -85,B 0,C 180,E1 -15128.848,E2 -15128.848} C_VEL
LIN {X 0,Y 319.674,Z 518.964,A -85,B 0,C 180,E1 -15132.7,E2 -15132.7} C_VEL
LIN {X 0,Y 319.688,Z 518.961,A -85,B 0,C 180,E1 -15135.295,E2 -15135.295} C_VEL
LIN {X 0,Y 319.681,Z 518.941,A -85,B 0,C 180,E1 -15139.254,E2 -15139.254} C_VEL
LIN {X 0,Y 319.625,Z 518.947,A -85,B 0,C 180,E1 -15143.315,E2 -15143.315} C_VEL
LIN {X 0,Y 319.626,Z 518.951,A -85,B 0,C 180,E1 -15146.088,E2 -15146.088} C_VEL
LIN {X 0,Y 319.579,Z 518.991,A -85,B 0,C 180,E1 -15148.934,E2 -15148.934} C_VEL
LIN {X 0,Y 319.583,Z 519.182,A -85,B 0,C 180,E1 -15151.081,E2 -15151.081} C_VEL
LIN {X 0,Y 321.153,Z 526.18,A -85,B 0,C 180,E1 -15154.678,E2 -15154.678} C_VEL
LIN {X 0,Y 322.811,Z 533.811,A -85,B 0,C 180,E1 -15158.396,E2 -15158.396} C_VEL
LIN {X 0,Y 324.206,Z 540.263,A -85,B 0,C 180,E1 -15161.388,E2 -15161.388} C_VEL
LIN {X 0,Y 325.705,Z 547.511,A -85,B 0,C 180,E1 -15164.599,E2 -15164.599} C_VEL
LIN {X 0,Y 326.797,Z 553.101,A -85,B 0,C 180,E1 -15166.986,E2 -15166.986} C_VEL
LIN {X 0,Y 326.96,Z 556.143,A -85,B 0,C 180,E1 -15168.217,E2 -15168.217} C_VEL
LIN {X 0,Y 326.629,Z 559.018,A -85,B 0,C 180,E1 -15169.298,E2 -15169.298} C_VEL
LIN {X 0,Y 327.694,Z 562.93,A -85,B 0,C 180,E1 -15169.606,E2 -15169.606} C_VEL
LIN {X 0,Y 328.716,Z 565.492,A -85,B 0,C 180,E1 -15169.859,E2 -15169.859} C_VEL
LIN {X 0,Y 333.743,Z 580.848,A -85,B 0,C 180,E1 -15171.182,E2 -15171.182} C_VEL
LIN {X 0,Y 337.744,Z 595.346,A -85,B 0,C 180,E1 -15172.432,E2 -15172.432} C_VEL
LIN {X 0,Y 340.585,Z 611.55,A -85,B 0,C 180,E1 -15173.8,E2 -15173.8} C_VEL
LIN {X 0,Y 342.461,Z 626.298,A -85,B 0,C 180,E1 -15175.172,E2 -15175.172} C_VEL
LIN {X 0,Y 343.291,Z 636.27,A -85,B 0,C 180,E1 -15176.157,E2 -15176.157} C_VEL
LIN {X 0,Y 340.469,Z 651.155,A -85,B 0,C 180,E1 -15177.368,E2 -15177.368} C_VEL
LIN {X 0,Y 337.513,Z 665.043,A -85,B 0,C 180,E1 -15178.745,E2 -15178.745} C_VEL
LIN {X 0,Y 334.386,Z 678.812,A -85,B 0,C 180,E1 -15180.404,E2 -15180.404} C_VEL
LIN {X 0,Y 331.436,Z 691.122,A -85,B 0,C 180,E1 -15182.194,E2 -15182.194} C_VEL
LIN {X 0,Y 328.388,Z 703.346,A -85,B 0,C 180,E1 -15184.301,E2 -15184.301} C_VEL
LIN {X 0,Y 325.721,Z 713.972,A -85,B 0,C 180,E1 -15186.475,E2 -15186.475} C_VEL
LIN {X 0,Y 323.242,Z 724.387,A -85,B 0,C 180,E1 -15189.025,E2 -15189.025} C_VEL
LIN {X 0,Y 321.414,Z 732.843,A -85,B 0,C 180,E1 -15191.517,E2 -15191.517} C_VEL
LIN {X 0,Y 319.917,Z 740.037,A -85,B 0,C 180,E1 -15194.063,E2 -15194.063} C_VEL
LIN {X 0,Y 318.984,Z 746.035,A -85,B 0,C 180,E1 -15196.626,E2 -15196.626} C_VEL
LIN {X 0,Y 318.296,Z 750.818,A -85,B 0,C 180,E1 -15199.184,E2 -15199.184} C_VEL
LIN {X 0,Y 318.079,Z 753.73,A -85,B 0,C 180,E1 -15201.104,E2 -15201.104} C_VEL
LIN {X 0,Y 318.078,Z 756.841,A -85,B 0,C 180,E1 -15203.866,E2 -15203.866} C_VEL
LIN {X 0,Y 317.983,Z 758.599,A -85,B 0,C 180,E1 -15206.2,E2 -15206.2} C_VEL
LIN {X 0,Y 318.177,Z 759.491,A -85,B 0,C 180,E1 -15208.736,E2 -15208.736} C_VEL
LIN {X 0,Y 318.202,Z 759.448,A -85,B 0,C 180,E1 -15211.267,E2 -15211.267} C_VEL
LIN {X 0,Y 317.996,Z 758.299,A -85,B 0,C 180,E1 -15213.803,E2 -15213.803} C_VEL
LIN {X 0,Y 318.092,Z 756.231,A -85,B 0,C 180,E1 -15216.344,E2 -15216.344} C_VEL
LIN {X 0,Y 318.123,Z 752.997,A -85,B 0,C 180,E1 -15218.897,E2 -15218.897} C_VEL
LIN {X 0,Y 318.466,Z 748.742,A -85,B 0,C 180,E1 -15221.457,E2 -15221.457} C_VEL
LIN {X 0,Y 319.301,Z 742.323,A -85,B 0,C 180,E1 -15224.429,E2 -15224.429} C_VEL
LIN {X 0,Y 320.542,Z 734.682,A -85,B 0,C 180,E1 -15227.218,E2 -15227.218} C_VEL
LIN {X 0,Y 322.177,Z 726.142,A -85,B 0,C 180,E1 -15229.763,E2 -15229.763} C_VEL
LIN {X 0,Y 324.232,Z 715.95,A -85,B 0,C 180,E1 -15232.293,E2 -15232.293} C_VEL
LIN {X 0,Y 326.538,Z 705.442,A -85,B 0,C 180,E1 -15234.477,E2 -15234.477} C_VEL
LIN {X 0,Y 328.909,Z 694.569,A -85,B 0,C 180,E1 -15236.398,E2 -15236.398} C_VEL
LIN {X 0,Y 331.42,Z 682.779,A -85,B 0,C 180,E1 -15238.154,E2 -15238.154} C_VEL
LIN {X 0,Y 336.228,Z 664.378,A -85,B 0,C 180,E1 -15240.811,E2 -15240.811} C_VEL
LIN {X 0,Y 340.757,Z 648.036,A -85,B 0,C 180,E1 -15242.78,E2 -15242.78} C_VEL
LIN {X 0,Y 343.862,Z 636.939,A -85,B 0,C 180,E1 -15243.925,E2 -15243.925} C_VEL
LIN {X 0,Y 344.875,Z 621.853,A -85,B 0,C 180,E1 -15245.866,E2 -15245.866} C_VEL
LIN {X 0,Y 345.961,Z 609.191,A -85,B 0,C 180,E1 -15247.398,E2 -15247.398} C_VEL
LIN {X 0,Y 346.241,Z 597.678,A -85,B 0,C 180,E1 -15248.995,E2 -15248.995} C_VEL
LIN {X 0,Y 346.14,Z 588.299,A -85,B 0,C 180,E1 -15250.522,E2 -15250.522} C_VEL
LIN {X 0,Y 345.97,Z 582.355,A -85,B 0,C 180,E1 -15251.673,E2 -15251.673} C_VEL
LIN {X 0,Y 345.892,Z 576.535,A -85,B 0,C 180,E1 -15252.991,E2 -15252.991} C_VEL
LIN {X 0,Y 345.972,Z 572.523,A -85,B 0,C 180,E1 -15254.065,E2 -15254.065} C_VEL
LIN {X 0,Y 345.77,Z 569.885,A -85,B 0,C 180,E1 -15255.35,E2 -15255.35} C_VEL
LIN {X 0,Y 346.09,Z 567.544,A -85,B 0,C 180,E1 -15256.975,E2 -15256.975} C_VEL
LIN {X 0,Y 346.915,Z 566.399,A -85,B 0,C 180,E1 -15258.554,E2 -15258.554} C_VEL
LIN {X 0,Y 348.116,Z 566.736,A -85,B 0,C 180,E1 -15260.101,E2 -15260.101} C_VEL
LIN {X 0,Y 349.806,Z 567.806,A -85,B 0,C 180,E1 -15261.588,E2 -15261.588} C_VEL
LIN {X 0,Y 351.844,Z 569.951,A -85,B 0,C 180,E1 -15263.035,E2 -15263.035} C_VEL
LIN {X 0,Y 354.001,Z 573.415,A -85,B 0,C 180,E1 -15264.487,E2 -15264.487} C_VEL
LIN {X 0,Y 354.683,Z 574.721,A -85,B 0,C 180,E1 -15264.927,E2 -15264.927} C_VEL
LIN {X 0,Y 354.544,Z 576.708,A -85,B 0,C 180,E1 -15265.238,E2 -15265.238} C_VEL
LIN {X 0,Y 350.029,Z 592.526,A -85,B 0,C 180,E1 -15266.83,E2 -15266.83} C_VEL
LIN {X 0,Y 345.529,Z 607.675,A -85,B 0,C 180,E1 -15268.681,E2 -15268.681} C_VEL
LIN {X 0,Y 341.147,Z 621.658,A -85,B 0,C 180,E1 -15270.708,E2 -15270.708} C_VEL
LIN {X 0,Y 337.336,Z 633.355,A -85,B 0,C 180,E1 -15272.72,E2 -15272.72} C_VEL
LIN {X 0,Y 333.59,Z 644.866,A -85,B 0,C 180,E1 -15275.08,E2 -15275.08} C_VEL
LIN {X 0,Y 330.263,Z 654.697,A -85,B 0,C 180,E1 -15277.478,E2 -15277.478} C_VEL
LIN {X 0,Y 327.462,Z 663.003,A -85,B 0,C 180,E1 -15279.917,E2 -15279.917} C_VEL
LIN {X 0,Y 325.138,Z 669.961,A -85,B 0,C 180,E1 -15282.386,E2 -15282.386} C_VEL
LIN {X 0,Y 323.206,Z 675.765,A -85,B 0,C 180,E1 -15284.875,E2 -15284.875} C_VEL
LIN {X 0,Y 321.75,Z 680.32,A -85,B 0,C 180,E1 -15287.384,E2 -15287.384} C_VEL
LIN {X 0,Y 320.635,Z 683.868,A -85,B 0,C 180,E1 -15289.901,E2 -15289.901} C_VEL
LIN {X 0,Y 319.912,Z 686.385,A -85,B 0,C 180,E1 -15292.426,E2 -15292.426} C_VEL
LIN {X 0,Y 319.303,Z 687.915,A -85,B 0,C 180,E1 -15294.95,E2 -15294.95} C_VEL
LIN {X 0,Y 318.798,Z 688.545,A -85,B 0,C 180,E1 -15297.474,E2 -15297.474} C_VEL
LIN {X 0,Y 318.571,Z 688.104,A -85,B 0,C 180,E1 -15300.001,E2 -15300.001} C_VEL
LIN {X 0,Y 318.758,Z 686.731,A -85,B 0,C 180,E1 -15302.528,E2 -15302.528} C_VEL
LIN {X 0,Y 318.946,Z 685.665,A -85,B 0,C 180,E1 -15303.791,E2 -15303.791} C_VEL
LIN {X 0,Y 318.925,Z 682.771,A -85,B 0,C 180,E1 -15306.326,E2 -15306.326} C_VEL
LIN {X 0,Y 319.361,Z 678.842,A -85,B 0,C 180,E1 -15308.862,E2 -15308.862} C_VEL
LIN {X 0,Y 319.887,Z 673.775,A -85,B 0,C 180,E1 -15311.405,E2 -15311.405} C_VEL
LIN {X 0,Y 320.771,Z 667.472,A -85,B 0,C 180,E1 -15313.947,E2 -15313.947} C_VEL
LIN {X 0,Y 322.009,Z 659.866,A -85,B 0,C 180,E1 -15316.484,E2 -15316.484} C_VEL
LIN {X 0,Y 323.589,Z 650.749,A -85,B 0,C 180,E1 -15319.014,E2 -15319.014} C_VEL
LIN {X 0,Y 325.593,Z 639.87,A -85,B 0,C 180,E1 -15321.528,E2 -15321.528} C_VEL
LIN {X 0,Y 327.602,Z 628.612,A -85,B 0,C 180,E1 -15323.719,E2 -15323.719} C_VEL
LIN {X 0,Y 329.692,Z 617.421,A -85,B 0,C 180,E1 -15325.574,E2 -15325.574} C_VEL
LIN {X 0,Y 332.217,Z 603.297,A -85,B 0,C 180,E1 -15327.571,E2 -15327.571} C_VEL
LIN {X 0,Y 334.741,Z 587.884,A -85,B 0,C 180,E1 -15329.392,E2 -15329.392} C_VEL
LIN {X 0,Y 337.195,Z 572.558,A -85,B 0,C 180,E1 -15330.881,E2 -15330.881} C_VEL
LIN {X 0,Y 338.227,Z 564.447,A -85,B 0,C 180,E1 -15331.576,E2 -15331.576} C_VEL
LIN {X 0,Y 337.75,Z 562.126,A -85,B 0,C 180,E1 -15331.827,E2 -15331.827} C_VEL
LIN {X 0,Y 332.551,Z 548.815,A -85,B 0,C 180,E1 -15333.405,E2 -15333.405} C_VEL
LIN {X 0,Y 326.213,Z 533.92,A -85,B 0,C 180,E1 -15335.046,E2 -15335.046} C_VEL
LIN {X 0,Y 319.702,Z 519.579,A -85,B 0,C 180,E1 -15336.518,E2 -15336.518} C_VEL
LIN {X 0,Y 319.604,Z 518.986,A -85,B 0,C 180,E1 -15336.618,E2 -15336.618} C_VEL
LIN {X 0,Y 319.564,Z 518.992,A -85,B 0,C 180,E1 -15339.669,E2 -15339.669} C_VEL
LIN {X 0,Y 319.527,Z 518.996,A -85,B 0,C 180,E1 -15343.46,E2 -15343.46} C_VEL
LIN {X 0,Y 319.56,Z 518.991,A -85,B 0,C 180,E1 -15347.016,E2 -15347.016} C_VEL
LIN {X 0,Y 319.553,Z 518.996,A -85,B 0,C 180,E1 -15350.371,E2 -15350.371} C_VEL
LIN {X 0,Y 319.565,Z 518.993,A -85,B 0,C 180,E1 -15353.572,E2 -15353.572} C_VEL
LIN {X 0,Y 319.625,Z 519.171,A -85,B 0,C 180,E1 -15357.225,E2 -15357.225} C_VEL
LIN {X 0,Y 320.515,Z 523.744,A -85,B 0,C 180,E1 -15360.437,E2 -15360.437} C_VEL
LIN {X 0,Y 321.115,Z 526.922,A -85,B 0,C 180,E1 -15362.637,E2 -15362.637} C_VEL
LIN {X 0,Y 321.41,Z 531.098,A -85,B 0,C 180,E1 -15365.451,E2 -15365.451} C_VEL
LIN {X 0,Y 321.413,Z 533.107,A -85,B 0,C 180,E1 -15366.69,E2 -15366.69} C_VEL
LIN {X 0,Y 322.794,Z 536.398,A -85,B 0,C 180,E1 -15366.949,E2 -15366.949} C_VEL
LIN {X 0,Y 330.102,Z 552.715,A -85,B 0,C 180,E1 -15368.332,E2 -15368.332} C_VEL
LIN {X 0,Y 335.6,Z 567.071,A -85,B 0,C 180,E1 -15369.618,E2 -15369.618} C_VEL
LIN {X 0,Y 340.33,Z 581.945,A -85,B 0,C 180,E1 -15371.042,E2 -15371.042} C_VEL
LIN {X 0,Y 342.368,Z 589.335,A -85,B 0,C 180,E1 -15371.791,E2 -15371.791} C_VEL
LIN {X 0,Y 340.361,Z 603.815,A -85,B 0,C 180,E1 -15372.833,E2 -15372.833} C_VEL
LIN {X 0,Y 337.976,Z 618.675,A -85,B 0,C 180,E1 -15374.16,E2 -15374.16} C_VEL
LIN {X 0,Y 335.359,Z 633.101,A -85,B 0,C 180,E1 -15375.744,E2 -15375.744} C_VEL
LIN {X 0,Y 332.609,Z 646.365,A -85,B 0,C 180,E1 -15377.491,E2 -15377.491} C_VEL
LIN {X 0,Y 329.876,Z 659.399,A -85,B 0,C 180,E1 -15379.565,E2 -15379.565} C_VEL
LIN {X 0,Y 327.371,Z 670.483,A -85,B 0,C 180,E1 -15381.667,E2 -15381.667} C_VEL
LIN {X 0,Y 325.196,Z 680.01,A -85,B 0,C 180,E1 -15383.795,E2 -15383.795} C_VEL
LIN {X 0,Y 323.043,Z 689.193,A -85,B 0,C 180,E1 -15386.257,E2 -15386.257} C_VEL
LIN {X 0,Y 321.412,Z 696.881,A -85,B 0,C 180,E1 -15388.746,E2 -15388.746} C_VEL
LIN {X 0,Y 320.12,Z 703.309,A -85,B 0,C 180,E1 -15391.257,E2 -15391.257} C_VEL
LIN {X 0,Y 319.254,Z 708.518,A -85,B 0,C 180,E1 -15393.785,E2 -15393.785} C_VEL
LIN {X 0,Y 318.507,Z 713.3,A -85,B 0,C 180,E1 -15396.805,E2 -15396.805} C_VEL
LIN {X 0,Y 318.152,Z 715.798,A -85,B 0,C 180,E1 -15398.894,E2 -15398.894} C_VEL
LIN {X 0,Y 317.892,Z 717.875,A -85,B 0,C 180,E1 -15401.475,E2 -15401.475} C_VEL
LIN {X 0,Y 317.812,Z 719.057,A -85,B 0,C 180,E1 -15404.077,E2 -15404.077} C_VEL
LIN {X 0,Y 317.787,Z 719.181,A -85,B 0,C 180,E1 -15406.707,E2 -15406.707} C_VEL
LIN {X 0,Y 317.958,Z 718.352,A -85,B 0,C 180,E1 -15409.361,E2 -15409.361} C_VEL
LIN {X 0,Y 318.352,Z 716.463,A -85,B 0,C 180,E1 -15412.041,E2 -15412.041} C_VEL
LIN {X 0,Y 318.99,Z 713.462,A -85,B 0,C 180,E1 -15414.745,E2 -15414.745} C_VEL
LIN {X 0,Y 320.002,Z 709.339,A -85,B 0,C 180,E1 -15417.463,E2 -15417.463} C_VEL
LIN {X 0,Y 321.29,Z 703.896,A -85,B 0,C 180,E1 -15420.204,E2 -15420.204} C_VEL
LIN {X 0,Y 323.113,Z 697.04,A -85,B 0,C 180,E1 -15422.939,E2 -15422.939} C_VEL
LIN {X 0,Y 325.477,Z 688.612,A -85,B 0,C 180,E1 -15425.66,E2 -15425.66} C_VEL
LIN {X 0,Y 328.095,Z 679.53,A -85,B 0,C 180,E1 -15428.076,E2 -15428.076} C_VEL
LIN {X 0,Y 330.655,Z 670.598,A -85,B 0,C 180,E1 -15430.077,E2 -15430.077} C_VEL
LIN {X 0,Y 333.381,Z 660.466,A -85,B 0,C 180,E1 -15432.012,E2 -15432.012} C_VEL
LIN {X 0,Y 336.622,Z 648.34,A -85,B 0,C 180,E1 -15433.961,E2 -15433.961} C_VEL
LIN {X 0,Y 339.861,Z 635.153,A -85,B 0,C 180,E1 -15435.732,E2 -15435.732} C_VEL
LIN {X 0,Y 342.635,Z 622.382,A -85,B 0,C 180,E1 -15437.16,E2 -15437.16} C_VEL
LIN {X 0,Y 345.048,Z 610.043,A -85,B 0,C 180,E1 -15438.325,E2 -15438.325} C_VEL
LIN {X 0,Y 345.239,Z 605.556,A -85,B 0,C 180,E1 -15438.788,E2 -15438.788} C_VEL
LIN {X 0,Y 344.393,Z 601.409,A -85,B 0,C 180,E1 -15439.326,E2 -15439.326} C_VEL
LIN {X 0,Y 341.811,Z 593.333,A -85,B 0,C 180,E1 -15440.461,E2 -15440.461} C_VEL
LIN {X 0,Y 338.542,Z 581.766,A -85,B 0,C 180,E1 -15441.922,E2 -15441.922} C_VEL
LIN {X 0,Y 333.745,Z 568.825,A -85,B 0,C 180,E1 -15443.588,E2 -15443.588} C_VEL
LIN {X 0,Y 327.657,Z 555.591,A -85,B 0,C 180,E1 -15445.36,E2 -15445.36} C_VEL
LIN {X 0,Y 323.194,Z 547.657,A -85,B 0,C 180,E1 -15446.51,E2 -15446.51} C_VEL
LIN {X 0,Y 321.052,Z 544.096,A -85,B 0,C 180,E1 -15447.054,E2 -15447.054} C_VEL
LIN {X 0,Y 318.484,Z 540.057,A -85,B 0,C 180,E1 -15447.689,E2 -15447.689} C_VEL
LIN {X 0,Y 316.264,Z 536.872,A -85,B 0,C 180,E1 -15448.242,E2 -15448.242} C_VEL
LIN {X 0,Y 315.737,Z 535.452,A -85,B 0,C 180,E1 -15448.429,E2 -15448.429} C_VEL
LIN {X 0,Y 315.03,Z 531.043,A -85,B 0,C 180,E1 -15452.063,E2 -15452.063} C_VEL
LIN {X 0,Y 314.434,Z 527.775,A -85,B 0,C 180,E1 -15454.869,E2 -15454.869} C_VEL
LIN {X 0,Y 313.699,Z 524.591,A -85,B 0,C 180,E1 -15457.612,E2 -15457.612} C_VEL
LIN {X 0,Y 312.664,Z 520.104,A -85,B 0,C 180,E1 -15461.657,E2 -15461.657} C_VEL
LIN {X 0,Y 312.618,Z 519.86,A -85,B 0,C 180,E1 -15462.332,E2 -15462.332} C_VEL
LIN {X 0,Y 312.685,Z 519.843,A -85,B 0,C 180,E1 -15465.685,E2 -15465.685} C_VEL
LIN {X 0,Y 312.694,Z 519.841,A -85,B 0,C 180,E1 -15469.641,E2 -15469.641} C_VEL
LIN {X 0,Y 312.863,Z 519.817,A -85,B 0,C 180,E1 -15472.253,E2 -15472.253} C_VEL
LIN {X 0,Y 312.713,Z 519.836,A -85,B 0,C 180,E1 -15474.842,E2 -15474.842} C_VEL
LIN {X 0,Y 312.944,Z 519.812,A -85,B 0,C 180,E1 -15477.425,E2 -15477.425} C_VEL
LIN {X 0,Y 313.111,Z 519.797,A -85,B 0,C 180,E1 -15479.999,E2 -15479.999} C_VEL
LIN {X 0,Y 312.929,Z 519.809,A -85,B 0,C 180,E1 -15482.574,E2 -15482.574} C_VEL
LIN {X 0,Y 312.899,Z 519.814,A -85,B 0,C 180,E1 -15486.448,E2 -15486.448} C_VEL
LIN {X 0,Y 312.777,Z 519.823,A -85,B 0,C 180,E1 -15489.049,E2 -15489.049} C_VEL
LIN {X 0,Y 312.626,Z 519.843,A -85,B 0,C 180,E1 -15492.991,E2 -15492.991} C_VEL
LIN {X 0,Y 312.627,Z 519.829,A -85,B 0,C 180,E1 -15495.65,E2 -15495.65} C_VEL
LIN {X 0,Y 312.625,Z 519.828,A -85,B 0,C 180,E1 -15499.706,E2 -15499.706} C_VEL
LIN {X 0,Y 312.58,Z 519.832,A -85,B 0,C 180,E1 -15502.809,E2 -15502.809} C_VEL
LIN {X 0,Y 312.545,Z 519.846,A -85,B 0,C 180,E1 -15506.726,E2 -15506.726} C_VEL
LIN {X 0,Y 312.571,Z 520.002,A -85,B 0,C 180,E1 -15510.391,E2 -15510.391} C_VEL
LIN {X 0,Y 314.403,Z 528.33,A -85,B 0,C 180,E1 -15514.75,E2 -15514.75} C_VEL
LIN {X 0,Y 316.254,Z 536.855,A -85,B 0,C 180,E1 -15518.944,E2 -15518.944} C_VEL
LIN {X 0,Y 317.78,Z 544.316,A -85,B 0,C 180,E1 -15522.412,E2 -15522.412} C_VEL
LIN {X 0,Y 319.338,Z 551.856,A -85,B 0,C 180,E1 -15525.76,E2 -15525.76} C_VEL
LIN {X 0,Y 320.035,Z 556.137,A -85,B 0,C 180,E1 -15527.591,E2 -15527.591} C_VEL
LIN {X 0,Y 320.009,Z 557.264,A -85,B 0,C 180,E1 -15528.038,E2 -15528.038} C_VEL
LIN {X 0,Y 321.147,Z 561.175,A -85,B 0,C 180,E1 -15528.377,E2 -15528.377} C_VEL
LIN {X 0,Y 322.169,Z 563.706,A -85,B 0,C 180,E1 -15528.646,E2 -15528.646} C_VEL
LIN {X 0,Y 327.483,Z 579.689,A -85,B 0,C 180,E1 -15530.116,E2 -15530.116} C_VEL
LIN {X 0,Y 331.697,Z 594.933,A -85,B 0,C 180,E1 -15531.493,E2 -15531.493} C_VEL
LIN {X 0,Y 334.593,Z 611.034,A -85,B 0,C 180,E1 -15532.921,E2 -15532.921} C_VEL
LIN {X 0,Y 336.385,Z 626.002,A -85,B 0,C 180,E1 -15534.351,E2 -15534.351} C_VEL
LIN {X 0,Y 337.319,Z 637.074,A -85,B 0,C 180,E1 -15535.493,E2 -15535.493} C_VEL
LIN {X 0,Y 334.523,Z 651.529,A -85,B 0,C 180,E1 -15536.713,E2 -15536.713} C_VEL
LIN {X 0,Y 331.29,Z 665.91,A -85,B 0,C 180,E1 -15538.18,E2 -15538.18} C_VEL
LIN {X 0,Y 328.207,Z 678.923,A -85,B 0,C 180,E1 -15539.789,E2 -15539.789} C_VEL
LIN {X 0,Y 325.116,Z 691.156,A -85,B 0,C 180,E1 -15541.605,E2 -15541.605} C_VEL
LIN {X 0,Y 321.848,Z 703.588,A -85,B 0,C 180,E1 -15543.807,E2 -15543.807} C_VEL
LIN {X 0,Y 318.776,Z 715.187,A -85,B 0,C 180,E1 -15546.276,E2 -15546.276} C_VEL
LIN {X 0,Y 316.539,Z 724.028,A -85,B 0,C 180,E1 -15548.512,E2 -15548.512} C_VEL
LIN {X 0,Y 314.568,Z 732.608,A -85,B 0,C 180,E1 -15551.099,E2 -15551.099} C_VEL
LIN {X 0,Y 312.985,Z 739.745,A -85,B 0,C 180,E1 -15553.701,E2 -15553.701} C_VEL
LIN {X 0,Y 311.991,Z 745.699,A -85,B 0,C 180,E1 -15556.32,E2 -15556.32} C_VEL
LIN {X 0,Y 311.264,Z 750.467,A -85,B 0,C 180,E1 -15558.937,E2 -15558.937} C_VEL
LIN {X 0,Y 310.993,Z 753.361,A -85,B 0,C 180,E1 -15560.9,E2 -15560.9} C_VEL
LIN {X 0,Y 311.007,Z 756.572,A -85,B 0,C 180,E1 -15563.871,E2 -15563.871} C_VEL
LIN {X 0,Y 310.91,Z 758.184,A -85,B 0,C 180,E1 -15566.113,E2 -15566.113} C_VEL
LIN {X 0,Y 311.08,Z 759.046,A -85,B 0,C 180,E1 -15568.707,E2 -15568.707} C_VEL
LIN {X 0,Y 311.122,Z 758.987,A -85,B 0,C 180,E1 -15571.296,E2 -15571.296} C_VEL
LIN {X 0,Y 310.926,Z 757.812,A -85,B 0,C 180,E1 -15573.89,E2 -15573.89} C_VEL
LIN {X 0,Y 310.988,Z 755.714,A -85,B 0,C 180,E1 -15576.489,E2 -15576.489} C_VEL
LIN {X 0,Y 311.122,Z 751.529,A -85,B 0,C 180,E1 -15579.755,E2 -15579.755} C_VEL
LIN {X 0,Y 311.758,Z 745.598,A -85,B 0,C 180,E1 -15583.029,E2 -15583.029} C_VEL
LIN {X 0,Y 312.662,Z 739.447,A -85,B 0,C 180,E1 -15585.65,E2 -15585.65} C_VEL
LIN {X 0,Y 314.046,Z 732.009,A -85,B 0,C 180,E1 -15588.26,E2 -15588.26} C_VEL
LIN {X 0,Y 315.792,Z 723.078,A -85,B 0,C 180,E1 -15590.861,E2 -15590.861} C_VEL
LIN {X 0,Y 318.174,Z 712.401,A -85,B 0,C 180,E1 -15593.429,E2 -15593.429} C_VEL
LIN {X 0,Y 320.679,Z 701.294,A -85,B 0,C 180,E1 -15595.649,E2 -15595.649} C_VEL
LIN {X 0,Y 323.25,Z 690.208,A -85,B 0,C 180,E1 -15597.518,E2 -15597.518} C_VEL
LIN {X 0,Y 327.826,Z 673.421,A -85,B 0,C 180,E1 -15600.253,E2 -15600.253} C_VEL
LIN {X 0,Y 332.18,Z 658.692,A -85,B 0,C 180,E1 -15602.292,E2 -15602.292} C_VEL
LIN {X 0,Y 336.805,Z 643.229,A -85,B 0,C 180,E1 -15604.112,E2 -15604.112} C_VEL
LIN {X 0,Y 338.242,Z 638.569,A -85,B 0,C 180,E1 -15604.605,E2 -15604.605} C_VEL
LIN {X 0,Y 339.403,Z 625.747,A -85,B 0,C 180,E1 -15606.352,E2 -15606.352} C_VEL
LIN {X 0,Y 341.157,Z 611.625,A -85,B 0,C 180,E1 -15608.172,E2 -15608.172} C_VEL
LIN {X 0,Y 341.878,Z 600.216,A -85,B 0,C 180,E1 -15609.867,E2 -15609.867} C_VEL
LIN {X 0,Y 342.148,Z 591.495,A -85,B 0,C 180,E1 -15611.396,E2 -15611.396} C_VEL
LIN {X 0,Y 342.417,Z 584.369,A -85,B 0,C 180,E1 -15612.901,E2 -15612.901} C_VEL
LIN {X 0,Y 342.84,Z 578.155,A -85,B 0,C 180,E1 -15614.574,E2 -15614.574} C_VEL
LIN {X 0,Y 342.985,Z 574.676,A -85,B 0,C 180,E1 -15616.563,E2 -15616.563} C_VEL
LIN {X 0,Y 343.351,Z 573.596,A -85,B 0,C 180,E1 -15617.51,E2 -15617.51} C_VEL
LIN {X 0,Y 344.378,Z 572.945,A -85,B 0,C 180,E1 -15619.229,E2 -15619.229} C_VEL
LIN {X 0,Y 345.949,Z 573.707,A -85,B 0,C 180,E1 -15620.968,E2 -15620.968} C_VEL
LIN {X 0,Y 347.319,Z 574.787,A -85,B 0,C 180,E1 -15622.109,E2 -15622.109} C_VEL
LIN {X 0,Y 349.219,Z 577.536,A -85,B 0,C 180,E1 -15623.611,E2 -15623.611} C_VEL
LIN {X 0,Y 350.267,Z 579.586,A -85,B 0,C 180,E1 -15624.418,E2 -15624.418} C_VEL
LIN {X 0,Y 345.202,Z 595.772,A -85,B 0,C 180,E1 -15626.129,E2 -15626.129} C_VEL
LIN {X 0,Y 340.678,Z 609.569,A -85,B 0,C 180,E1 -15627.874,E2 -15627.874} C_VEL
LIN {X 0,Y 336.095,Z 622.989,A -85,B 0,C 180,E1 -15629.878,E2 -15629.878} C_VEL
LIN {X 0,Y 331.477,Z 636.042,A -85,B 0,C 180,E1 -15632.197,E2 -15632.197} C_VEL
LIN {X 0,Y 327.525,Z 647.165,A -85,B 0,C 180,E1 -15634.586,E2 -15634.586} C_VEL
LIN {X 0,Y 323.99,Z 656.692,A -85,B 0,C 180,E1 -15637.018,E2 -15637.018} C_VEL
LIN {X 0,Y 321.035,Z 664.764,A -85,B 0,C 180,E1 -15639.497,E2 -15639.497} C_VEL
LIN {X 0,Y 318.551,Z 671.562,A -85,B 0,C 180,E1 -15642.009,E2 -15642.009} C_VEL
LIN {X 0,Y 316.492,Z 677.182,A -85,B 0,C 180,E1 -15644.546,E2 -15644.546} C_VEL
LIN {X 0,Y 314.932,Z 681.65,A -85,B 0,C 180,E1 -15647.106,E2 -15647.106} C_VEL
LIN {X 0,Y 313.46,Z 686.05,A -85,B 0,C 180,E1 -15650.582,E2 -15650.582} C_VEL
LIN {X 0,Y 312.594,Z 688.323,A -85,B 0,C 180,E1 -15653.546,E2 -15653.546} C_VEL
LIN {X 0,Y 312.005,Z 689.294,A -85,B 0,C 180,E1 -15656.126,E2 -15656.126} C_VEL
LIN {X 0,Y 311.602,Z 689.331,A -85,B 0,C 180,E1 -15658.708,E2 -15658.708} C_VEL
LIN {X 0,Y 311.564,Z 688.316,A -85,B 0,C 180,E1 -15661.293,E2 -15661.293} C_VEL
LIN {X 0,Y 311.896,Z 686.37,A -85,B 0,C 180,E1 -15663.877,E2 -15663.877} C_VEL
LIN {X 0,Y 311.884,Z 683.374,A -85,B 0,C 180,E1 -15666.47,E2 -15666.47} C_VEL
LIN {X 0,Y 312.346,Z 679.341,A -85,B 0,C 180,E1 -15669.063,E2 -15669.063} C_VEL
LIN {X 0,Y 312.915,Z 674.188,A -85,B 0,C 180,E1 -15671.663,E2 -15671.663} C_VEL
LIN {X 0,Y 313.863,Z 667.766,A -85,B 0,C 180,E1 -15674.26,E2 -15674.26} C_VEL
LIN {X 0,Y 315.117,Z 660.016,A -85,B 0,C 180,E1 -15676.855,E2 -15676.855} C_VEL
LIN {X 0,Y 316.803,Z 650.753,A -85,B 0,C 180,E1 -15679.437,E2 -15679.437} C_VEL
LIN {X 0,Y 318.893,Z 639.723,A -85,B 0,C 180,E1 -15682.004,E2 -15682.004} C_VEL
LIN {X 0,Y 321.009,Z 628.372,A -85,B 0,C 180,E1 -15684.237,E2 -15684.237} C_VEL
LIN {X 0,Y 323.586,Z 615.017,A -85,B 0,C 180,E1 -15686.439,E2 -15686.439} C_VEL
LIN {X 0,Y 326.279,Z 600.366,A -85,B 0,C 180,E1 -15688.462,E2 -15688.462} C_VEL
LIN {X 0,Y 328.685,Z 585.65,A -85,B 0,C 180,E1 -15690.165,E2 -15690.165} C_VEL
LIN {X 0,Y 330.98,Z 571.461,A -85,B 0,C 180,E1 -15691.528,E2 -15691.528} C_VEL
LIN {X 0,Y 331.679,Z 565.528,A -85,B 0,C 180,E1 -15692.051,E2 -15692.051} C_VEL
LIN {X 0,Y 325.885,Z 550.625,A -85,B 0,C 180,E1 -15693.872,E2 -15693.872} C_VEL
LIN {X 0,Y 319.646,Z 535.89,A -85,B 0,C 180,E1 -15695.558,E2 -15695.558} C_VEL
LIN {X 0,Y 313.376,Z 522.372,A -85,B 0,C 180,E1 -15697.026,E2 -15697.026} C_VEL
LIN {X 0,Y 312.578,Z 519.863,A -85,B 0,C 180,E1 -15697.273,E2 -15697.273} C_VEL
LIN {X 0,Y 312.496,Z 519.874,A -85,B 0,C 180,E1 -15700.709,E2 -15700.709} C_VEL
LIN {X 0,Y 312.457,Z 519.878,A -85,B 0,C 180,E1 -15704.21,E2 -15704.21} C_VEL
LIN {X 0,Y 312.49,Z 519.873,A -85,B 0,C 180,E1 -15707.918,E2 -15707.918} C_VEL
LIN {X 0,Y 312.541,Z 519.87,A -85,B 0,C 180,E1 -15711.91,E2 -15711.91} C_VEL
LIN {X 0,Y 312.512,Z 519.873,A -85,B 0,C 180,E1 -15715.79,E2 -15715.79} C_VEL
LIN {X 0,Y 312.539,Z 519.908,A -85,B 0,C 180,E1 -15716.427,E2 -15716.427} C_VEL
LIN {X 0,Y 313.481,Z 524.52,A -85,B 0,C 180,E1 -15719.705,E2 -15719.705} C_VEL
LIN {X 0,Y 314.242,Z 528.79,A -85,B 0,C 180,E1 -15722.71,E2 -15722.71} C_VEL
LIN {X 0,Y 314.508,Z 533.344,A -85,B 0,C 180,E1 -15725.825,E2 -15725.825} C_VEL
LIN {X 0,Y 315.911,Z 536.723,A -85,B 0,C 180,E1 -15726.102,E2 -15726.102} C_VEL
LIN {X 0,Y 323.073,Z 552.474,A -85,B 0,C 180,E1 -15727.498,E2 -15727.498} C_VEL
LIN {X 0,Y 328.703,Z 566.97,A -85,B 0,C 180,E1 -15728.848,E2 -15728.848} C_VEL
LIN {X 0,Y 333.359,Z 581.621,A -85,B 0,C 180,E1 -15730.285,E2 -15730.285} C_VEL
LIN {X 0,Y 335.839,Z 590.265,A -85,B 0,C 180,E1 -15731.198,E2 -15731.198} C_VEL
LIN {X 0,Y 335.783,Z 593.119,A -85,B 0,C 180,E1 -15731.421,E2 -15731.421} C_VEL
LIN {X 0,Y 333.59,Z 607.76,A -85,B 0,C 180,E1 -15732.554,E2 -15732.554} C_VEL
LIN {X 0,Y 331.012,Z 622.692,A -85,B 0,C 180,E1 -15733.976,E2 -15733.976} C_VEL
LIN {X 0,Y 328.363,Z 636.6,A -85,B 0,C 180,E1 -15735.592,E2 -15735.592} C_VEL
LIN {X 0,Y 325.839,Z 648.446,A -85,B 0,C 180,E1 -15737.226,E2 -15737.226} C_VEL
LIN {X 0,Y 323.389,Z 659.504,A -85,B 0,C 180,E1 -15739.037,E2 -15739.037} C_VEL
LIN {X 0,Y 320.773,Z 670.646,A -85,B 0,C 180,E1 -15741.177,E2 -15741.177} C_VEL
LIN {X 0,Y 318.507,Z 680.203,A -85,B 0,C 180,E1 -15743.346,E2 -15743.346} C_VEL
LIN {X 0,Y 316.258,Z 689.427,A -85,B 0,C 180,E1 -15745.857,E2 -15745.857} C_VEL
LIN {X 0,Y 314.727,Z 696.277,A -85,B 0,C 180,E1 -15748.079,E2 -15748.079} C_VEL
LIN {X 0,Y 313.347,Z 702.895,A -85,B 0,C 180,E1 -15750.641,E2 -15750.641} C_VEL
LIN {X 0,Y 312.152,Z 709.463,A -85,B 0,C 180,E1 -15753.872,E2 -15753.872} C_VEL
LIN {X 0,Y 311.423,Z 713.889,A -85,B 0,C 180,E1 -15756.796,E2 -15756.796} C_VEL
LIN {X 0,Y 311.042,Z 716.503,A -85,B 0,C 180,E1 -15759.099,E2 -15759.099} C_VEL
LIN {X 0,Y 310.803,Z 718.492,A -85,B 0,C 180,E1 -15761.741,E2 -15761.741} C_VEL
LIN {X 0,Y 310.724,Z 719.547,A -85,B 0,C 180,E1 -15764.405,E2 -15764.405} C_VEL
LIN {X 0,Y 310.739,Z 719.608,A -85,B 0,C 180,E1 -15767.097,E2 -15767.097} C_VEL
LIN {X 0,Y 310.933,Z 718.649,A -85,B 0,C 180,E1 -15769.817,E2 -15769.817} C_VEL
LIN {X 0,Y 311.368,Z 716.695,A -85,B 0,C 180,E1 -15772.562,E2 -15772.562} C_VEL
LIN {X 0,Y 312.291,Z 712.919,A -85,B 0,C 180,E1 -15775.816,E2 -15775.816} C_VEL
LIN {X 0,Y 313.203,Z 709.279,A -85,B 0,C 180,E1 -15778.112,E2 -15778.112} C_VEL
LIN {X 0,Y 314.665,Z 703.75,A -85,B 0,C 180,E1 -15780.909,E2 -15780.909} C_VEL
LIN {X 0,Y 316.664,Z 696.74,A -85,B 0,C 180,E1 -15783.698,E2 -15783.698} C_VEL
LIN {X 0,Y 319.21,Z 688.136,A -85,B 0,C 180,E1 -15786.472,E2 -15786.472} C_VEL
LIN {X 0,Y 321.926,Z 679.232,A -85,B 0,C 180,E1 -15788.834,E2 -15788.834} C_VEL
LIN {X 0,Y 325.07,Z 668.707,A -85,B 0,C 180,E1 -15791.17,E2 -15791.17} C_VEL
LIN {X 0,Y 328.352,Z 657.206,A -85,B 0,C 180,E1 -15793.303,E2 -15793.303} C_VEL
LIN {X 0,Y 331.707,Z 644.764,A -85,B 0,C 180,E1 -15795.214,E2 -15795.214} C_VEL
LIN {X 0,Y 334.818,Z 632.157,A -85,B 0,C 180,E1 -15796.835,E2 -15796.835} C_VEL
LIN {X 0,Y 337.795,Z 618.947,A -85,B 0,C 180,E1 -15798.257,E2 -15798.257} C_VEL
LIN {X 0,Y 340.548,Z 604.576,A -85,B 0,C 180,E1 -15799.55,E2 -15799.55} C_VEL
LIN {X 0,Y 342.179,Z 594.99,A -85,B 0,C 180,E1 -15800.262,E2 -15800.262} C_VEL
LIN {X 0,Y 341.811,Z 593.333,A -85,B 0,C 180,E1 -15800.461,E2 -15800.461} C_VEL
LIN {X 0,Y 340.06,Z 589.132,A -85,B 0,C 180,E1 -15801.096,E2 -15801.096} C_VEL
LIN {X 0,Y 335.686,Z 583.31,A -85,B 0,C 180,E1 -15802.241,E2 -15802.241} C_VEL
LIN {X 0,Y 332.04,Z 578.778,A -85,B 0,C 180,E1 -15803.184,E2 -15803.184} C_VEL
LIN {X 0,Y 329.704,Z 574.886,A -85,B 0,C 180,E1 -15803.854,E2 -15803.854} C_VEL
LIN {X 0,Y 329.091,Z 573.429,A -85,B 0,C 180,E1 -15804.064,E2 -15804.064} C_VEL
LIN {X 0,Y 323.397,Z 560.44,A -85,B 0,C 180,E1 -15805.878,E2 -15805.878} C_VEL
LIN {X 0,Y 319.207,Z 552.63,A -85,B 0,C 180,E1 -15807.064,E2 -15807.064} C_VEL
LIN {X 0,Y 316.995,Z 548.933,A -85,B 0,C 180,E1 -15807.654,E2 -15807.654} C_VEL
LIN {X 0,Y 314.464,Z 544.944,A -85,B 0,C 180,E1 -15808.329,E2 -15808.329} C_VEL
LIN {X 0,Y 311.604,Z 540.608,A -85,B 0,C 180,E1 -15809.081,E2 -15809.081} C_VEL
LIN {X 0,Y 309.459,Z 537.775,A -85,B 0,C 180,E1 -15809.647,E2 -15809.647} C_VEL
LIN {X 0,Y 308.749,Z 536.06,A -85,B 0,C 180,E1 -15809.877,E2 -15809.877} C_VEL
LIN {X 0,Y 308.181,Z 532.547,A -85,B 0,C 180,E1 -15812.864,E2 -15812.864} C_VEL
LIN {X 0,Y 307.466,Z 528.885,A -85,B 0,C 180,E1 -15816.103,E2 -15816.103} C_VEL
LIN {X 0,Y 306.519,Z 524.587,A -85,B 0,C 180,E1 -15820.057,E2 -15820.057} C_VEL
LIN {X 0,Y 305.585,Z 520.727,A -85,B 0,C 180,E1 -15823.979,E2 -15823.979} C_VEL
LIN {X 0,Y 305.581,Z 520.727,A -85,B 0,C 180,E1 -15826.703,E2 -15826.703} C_VEL
LIN {X 0,Y 305.787,Z 520.702,A -85,B 0,C 180,E1 -15831.206,E2 -15831.206} C_VEL
LIN {X 0,Y 305.845,Z 520.702,A -85,B 0,C 180,E1 -15833.402,E2 -15833.402} C_VEL
LIN {X 0,Y 305.89,Z 520.691,A -85,B 0,C 180,E1 -15837.366,E2 -15837.366} C_VEL
LIN {X 0,Y 306.064,Z 520.675,A -85,B 0,C 180,E1 -15839.999,E2 -15839.999} C_VEL
LIN {X 0,Y 305.878,Z 520.687,A -85,B 0,C 180,E1 -15842.633,E2 -15842.633} C_VEL
LIN {X 0,Y 305.842,Z 520.694,A -85,B 0,C 180,E1 -15846.597,E2 -15846.597} C_VEL
LIN {X 0,Y 305.725,Z 520.701,A -85,B 0,C 180,E1 -15849.259,E2 -15849.259} C_VEL
LIN {X 0,Y 305.58,Z 520.723,A -85,B 0,C 180,E1 -15853.296,E2 -15853.296} C_VEL
LIN {X 0,Y 305.583,Z 520.697,A -85,B 0,C 180,E1 -15856.02,E2 -15856.02} C_VEL
LIN {X 0,Y 305.604,Z 520.696,A -85,B 0,C 180,E1 -15859.465,E2 -15859.465} C_VEL
LIN {X 0,Y 305.545,Z 520.702,A -85,B 0,C 180,E1 -15863.07,E2 -15863.07} C_VEL
LIN {X 0,Y 305.539,Z 520.706,A -85,B 0,C 180,E1 -15866.228,E2 -15866.228} C_VEL
LIN {X 0,Y 305.522,Z 520.777,A -85,B 0,C 180,E1 -15869.659,E2 -15869.659} C_VEL
LIN {X 0,Y 307.264,Z 528.855,A -85,B 0,C 180,E1 -15873.992,E2 -15873.992} C_VEL
LIN {X 0,Y 308.932,Z 536.568,A -85,B 0,C 180,E1 -15877.895,E2 -15877.895} C_VEL
LIN {X 0,Y 310.612,Z 544.508,A -85,B 0,C 180,E1 -15881.7,E2 -15881.7} C_VEL
LIN {X 0,Y 312.468,Z 553.547,A -85,B 0,C 180,E1 -15885.796,E2 -15885.796} C_VEL
LIN {X 0,Y 312.795,Z 555.268,A -85,B 0,C 180,E1 -15886.552,E2 -15886.552} C_VEL
LIN {X 0,Y 314.288,Z 559.315,A -85,B 0,C 180,E1 -15886.995,E2 -15886.995} C_VEL
LIN {X 0,Y 315.751,Z 562.205,A -85,B 0,C 180,E1 -15887.384,E2 -15887.384} C_VEL
LIN {X 0,Y 317.929,Z 568.521,A -85,B 0,C 180,E1 -15888.013,E2 -15888.013} C_VEL
LIN {X 0,Y 322.35,Z 581.91,A -85,B 0,C 180,E1 -15889.309,E2 -15889.309} C_VEL
LIN {X 0,Y 326.544,Z 598.112,A -85,B 0,C 180,E1 -15890.855,E2 -15890.855} C_VEL
LIN {X 0,Y 328.972,Z 612.858,A -85,B 0,C 180,E1 -15892.227,E2 -15892.227} C_VEL
LIN {X 0,Y 330.718,Z 629.216,A -85,B 0,C 180,E1 -15893.854,E2 -15893.854} C_VEL
LIN {X 0,Y 331.329,Z 639.201,A -85,B 0,C 180,E1 -15894.931,E2 -15894.931} C_VEL
LIN {X 0,Y 327.964,Z 655.027,A -85,B 0,C 180,E1 -15896.327,E2 -15896.327} C_VEL
LIN {X 0,Y 324.714,Z 668.576,A -85,B 0,C 180,E1 -15897.806,E2 -15897.806} C_VEL
LIN {X 0,Y 321.199,Z 682.21,A -85,B 0,C 180,E1 -15899.605,E2 -15899.605} C_VEL
LIN {X 0,Y 317.851,Z 694.845,A -85,B 0,C 180,E1 -15901.617,E2 -15901.617} C_VEL
LIN {X 0,Y 314.641,Z 706.477,A -85,B 0,C 180,E1 -15903.825,E2 -15903.825} C_VEL
LIN {X 0,Y 311.47,Z 717.741,A -85,B 0,C 180,E1 -15906.392,E2 -15906.392} C_VEL
LIN {X 0,Y 308.976,Z 727.141,A -85,B 0,C 180,E1 -15908.988,E2 -15908.988} C_VEL
LIN {X 0,Y 307.251,Z 734.244,A -85,B 0,C 180,E1 -15911.325,E2 -15911.325} C_VEL
LIN {X 0,Y 305.744,Z 741.102,A -85,B 0,C 180,E1 -15913.99,E2 -15913.99} C_VEL
LIN {X 0,Y 304.568,Z 747.919,A -85,B 0,C 180,E1 -15917.339,E2 -15917.339} C_VEL
LIN {X 0,Y 303.922,Z 752.995,A -85,B 0,C 180,E1 -15920.686,E2 -15920.686} C_VEL
LIN {X 0,Y 303.908,Z 756.347,A -85,B 0,C 180,E1 -15923.925,E2 -15923.925} C_VEL
LIN {X 0,Y 303.839,Z 757.766,A -85,B 0,C 180,E1 -15926.022,E2 -15926.022} C_VEL
LIN {X 0,Y 303.985,Z 758.601,A -85,B 0,C 180,E1 -15928.677,E2 -15928.677} C_VEL
LIN {X 0,Y 304.028,Z 758.52,A -85,B 0,C 180,E1 -15931.326,E2 -15931.326} C_VEL
LIN {X 0,Y 303.858,Z 757.321,A -85,B 0,C 180,E1 -15933.98,E2 -15933.98} C_VEL
LIN {X 0,Y 303.905,Z 755.189,A -85,B 0,C 180,E1 -15936.641,E2 -15936.641} C_VEL
LIN {X 0,Y 304.057,Z 750.974,A -85,B 0,C 180,E1 -15939.984,E2 -15939.984} C_VEL
LIN {X 0,Y 304.758,Z 745.005,A -85,B 0,C 180,E1 -15943.334,E2 -15943.334} C_VEL
LIN {X 0,Y 305.698,Z 738.819,A -85,B 0,C 180,E1 -15946.016,E2 -15946.016} C_VEL
LIN {X 0,Y 307.19,Z 731.329,A -85,B 0,C 180,E1 -15948.682,E2 -15948.682} C_VEL
LIN {X 0,Y 309.032,Z 722.335,A -85,B 0,C 180,E1 -15951.339,E2 -15951.339} C_VEL
LIN {X 0,Y 311.507,Z 711.592,A -85,B 0,C 180,E1 -15953.961,E2 -15953.961} C_VEL
LIN {X 0,Y 314.177,Z 700.459,A -85,B 0,C 180,E1 -15956.22,E2 -15956.22} C_VEL
LIN {X 0,Y 320.545,Z 677.842,A -85,B 0,C 180,E1 -15960.285,E2 -15960.285} C_VEL
LIN {X 0,Y 325.547,Z 662.014,A -85,B 0,C 180,E1 -15962.665,E2 -15962.665} C_VEL
LIN {X 0,Y 330.723,Z 646.289,A -85,B 0,C 180,E1 -15964.643,E2 -15964.643} C_VEL
LIN {X 0,Y 332.67,Z 640.257,A -85,B 0,C 180,E1 -15965.315,E2 -15965.315} C_VEL
LIN {X 0,Y 334.36,Z 627.123,A -85,B 0,C 180,E1 -15967.207,E2 -15967.207} C_VEL
LIN {X 0,Y 336.44,Z 614.023,A -85,B 0,C 180,E1 -15968.984,E2 -15968.984} C_VEL
LIN {X 0,Y 337.647,Z 602.632,A -85,B 0,C 180,E1 -15970.795,E2 -15970.795} C_VEL
LIN {X 0,Y 338.474,Z 593.592,A -85,B 0,C 180,E1 -15972.529,E2 -15972.529} C_VEL
LIN {X 0,Y 339.109,Z 587.449,A -85,B 0,C 180,E1 -15973.989,E2 -15973.989} C_VEL
LIN {X 0,Y 339.487,Z 584.84,A -85,B 0,C 180,E1 -15974.739,E2 -15974.739} C_VEL
LIN {X 0,Y 339.672,Z 583.356,A -85,B 0,C 180,E1 -15975.294,E2 -15975.294} C_VEL
LIN {X 0,Y 340.066,Z 580.711,A -85,B 0,C 180,E1 -15977.001,E2 -15977.001} C_VEL
LIN {X 0,Y 340.881,Z 579.456,A -85,B 0,C 180,E1 -15978.72,E2 -15978.72} C_VEL
LIN {X 0,Y 342.183,Z 579.719,A -85,B 0,C 180,E1 -15980.454,E2 -15980.454} C_VEL
LIN {X 0,Y 344.067,Z 581.242,A -85,B 0,C 180,E1 -15982.209,E2 -15982.209} C_VEL
LIN {X 0,Y 345.332,Z 583.287,A -85,B 0,C 180,E1 -15983.353,E2 -15983.353} C_VEL
LIN {X 0,Y 345.441,Z 585.131,A -85,B 0,C 180,E1 -15983.843,E2 -15983.843} C_VEL
LIN {X 0,Y 340.486,Z 599.297,A -85,B 0,C 180,E1 -15985.416,E2 -15985.416} C_VEL
LIN {X 0,Y 335.215,Z 613.775,A -85,B 0,C 180,E1 -15987.346,E2 -15987.346} C_VEL
LIN {X 0,Y 329.869,Z 627.891,A -85,B 0,C 180,E1 -15989.603,E2 -15989.603} C_VEL
LIN {X 0,Y 325.093,Z 640.165,A -85,B 0,C 180,E1 -15991.953,E2 -15991.953} C_VEL
LIN {X 0,Y 320.907,Z 650.831,A -85,B 0,C 180,E1 -15994.402,E2 -15994.402} C_VEL
LIN {X 0,Y 317.298,Z 659.816,A -85,B 0,C 180,E1 -15996.85,E2 -15996.85} C_VEL
LIN {X 0,Y 313.921,Z 668.371,A -85,B 0,C 180,E1 -15999.696,E2 -15999.696} C_VEL
LIN {X 0,Y 311.419,Z 674.696,A -85,B 0,C 180,E1 -16002.263,E2 -16002.263} C_VEL
LIN {X 0,Y 308.891,Z 680.978,A -85,B 0,C 180,E1 -16005.507,E2 -16005.507} C_VEL
LIN {X 0,Y 307.401,Z 684.774,A -85,B 0,C 180,E1 -16008.126,E2 -16008.126} C_VEL
LIN {X 0,Y 306.389,Z 687.556,A -85,B 0,C 180,E1 -16010.761,E2 -16010.761} C_VEL
LIN {X 0,Y 305.63,Z 689.396,A -85,B 0,C 180,E1 -16013.398,E2 -16013.398} C_VEL
LIN {X 0,Y 304.987,Z 690.255,A -85,B 0,C 180,E1 -16016.037,E2 -16016.037} C_VEL
LIN {X 0,Y 304.561,Z 690.211,A -85,B 0,C 180,E1 -16018.678,E2 -16018.678} C_VEL
LIN {X 0,Y 304.525,Z 689.091,A -85,B 0,C 180,E1 -16021.323,E2 -16021.323} C_VEL
LIN {X 0,Y 304.833,Z 687.035,A -85,B 0,C 180,E1 -16023.967,E2 -16023.967} C_VEL
LIN {X 0,Y 304.849,Z 683.971,A -85,B 0,C 180,E1 -16026.62,E2 -16026.62} C_VEL
LIN {X 0,Y 305.338,Z 679.818,A -85,B 0,C 180,E1 -16029.272,E2 -16029.272} C_VEL
LIN {X 0,Y 305.93,Z 674.593,A -85,B 0,C 180,E1 -16031.933,E2 -16031.933} C_VEL
LIN {X 0,Y 306.943,Z 668.041,A -85,B 0,C 180,E1 -16034.588,E2 -16034.588} C_VEL
LIN {X 0,Y 308.263,Z 660.155,A -85,B 0,C 180,E1 -16037.241,E2 -16037.241} C_VEL
LIN {X 0,Y 310.022,Z 650.74,A -85,B 0,C 180,E1 -16039.88,E2 -16039.88} C_VEL
LIN {X 0,Y 311.938,Z 641.079,A -85,B 0,C 180,E1 -16042.172,E2 -16042.172} C_VEL
LIN {X 0,Y 314.076,Z 629.767,A -85,B 0,C 180,E1 -16044.455,E2 -16044.455} C_VEL
LIN {X 0,Y 316.502,Z 617.515,A -85,B 0,C 180,E1 -16046.544,E2 -16046.544} C_VEL
LIN {X 0,Y 319.083,Z 604.02,A -85,B 0,C 180,E1 -16048.498,E2 -16048.498} C_VEL
LIN {X 0,Y 321.701,Z 588.878,A -85,B 0,C 180,E1 -16050.345,E2 -16050.345} C_VEL
LIN {X 0,Y 324.379,Z 572.935,A -85,B 0,C 180,E1 -16051.943,E2 -16051.943} C_VEL
LIN {X 0,Y 324.932,Z 567.176,A -85,B 0,C 180,E1 -16052.483,E2 -16052.483} C_VEL
LIN {X 0,Y 318.761,Z 551.115,A -85,B 0,C 180,E1 -16054.508,E2 -16054.508} C_VEL
LIN {X 0,Y 312.402,Z 536.169,A -85,B 0,C 180,E1 -16056.276,E2 -16056.276} C_VEL
LIN {X 0,Y 305.648,Z 521.506,A -85,B 0,C 180,E1 -16057.894,E2 -16057.894} C_VEL
LIN {X 0,Y 305.505,Z 520.743,A -85,B 0,C 180,E1 -16057.993,E2 -16057.993} C_VEL
LIN {X 0,Y 305.446,Z 520.75,A -85,B 0,C 180,E1 -16061.857,E2 -16061.857} C_VEL
LIN {X 0,Y 305.406,Z 520.755,A -85,B 0,C 180,E1 -16065.511,E2 -16065.511} C_VEL
LIN {X 0,Y 305.447,Z 520.75,A -85,B 0,C 180,E1 -16068.143,E2 -16068.143} C_VEL
LIN {X 0,Y 305.501,Z 520.746,A -85,B 0,C 180,E1 -16071.6,E2 -16071.6} C_VEL
LIN {X 0,Y 305.483,Z 520.823,A -85,B 0,C 180,E1 -16075.68,E2 -16075.68} C_VEL
LIN {X 0,Y 306.643,Z 526.38,A -85,B 0,C 180,E1 -16079.719,E2 -16079.719} C_VEL
LIN {X 0,Y 307.402,Z 531.098,A -85,B 0,C 180,E1 -16083.082,E2 -16083.082} C_VEL
LIN {X 0,Y 307.645,Z 533.955,A -85,B 0,C 180,E1 -16084.937,E2 -16084.937} C_VEL
LIN {X 0,Y 308.996,Z 537.047,A -85,B 0,C 180,E1 -16085.208,E2 -16085.208} C_VEL
LIN {X 0,Y 316.168,Z 552.429,A -85,B 0,C 180,E1 -16086.645,E2 -16086.645} C_VEL
LIN {X 0,Y 322.008,Z 567.43,A -85,B 0,C 180,E1 -16088.096,E2 -16088.096} C_VEL
LIN {X 0,Y 326.541,Z 581.439,A -85,B 0,C 180,E1 -16089.52,E2 -16089.52} C_VEL
LIN {X 0,Y 329.716,Z 592.723,A -85,B 0,C 180,E1 -16090.748,E2 -16090.748} C_VEL
LIN {X 0,Y 327.548,Z 607.196,A -85,B 0,C 180,E1 -16091.872,E2 -16091.872} C_VEL
LIN {X 0,Y 325.13,Z 621.161,A -85,B 0,C 180,E1 -16093.194,E2 -16093.194} C_VEL
LIN {X 0,Y 322.339,Z 635.413,A -85,B 0,C 180,E1 -16094.832,E2 -16094.832} C_VEL
LIN {X 0,Y 319.436,Z 648.453,A -85,B 0,C 180,E1 -16096.642,E2 -16096.642} C_VEL
LIN {X 0,Y 316.923,Z 659.582,A -85,B 0,C 180,E1 -16098.486,E2 -16098.486} C_VEL
LIN {X 0,Y 314.192,Z 670.796,A -85,B 0,C 180,E1 -16100.666,E2 -16100.666} C_VEL
LIN {X 0,Y 311.672,Z 681.055,A -85,B 0,C 180,E1 -16103.044,E2 -16103.044} C_VEL
LIN {X 0,Y 309.215,Z 690.75,A -85,B 0,C 180,E1 -16105.762,E2 -16105.762} C_VEL
LIN {X 0,Y 307.665,Z 697.433,A -85,B 0,C 180,E1 -16108.035,E2 -16108.035} C_VEL
LIN {X 0,Y 306.248,Z 703.935,A -85,B 0,C 180,E1 -16110.656,E2 -16110.656} C_VEL
LIN {X 0,Y 305.216,Z 709.189,A -85,B 0,C 180,E1 -16113.299,E2 -16113.299} C_VEL
LIN {X 0,Y 304.637,Z 712.459,A -85,B 0,C 180,E1 -16115.293,E2 -16115.293} C_VEL
LIN {X 0,Y 304.112,Z 715.837,A -85,B 0,C 180,E1 -16117.969,E2 -16117.969} C_VEL
LIN {X 0,Y 303.773,Z 718.297,A -85,B 0,C 180,E1 -16120.665,E2 -16120.665} C_VEL
LIN {X 0,Y 303.695,Z 719.763,A -85,B 0,C 180,E1 -16123.6,E2 -16123.6} C_VEL
LIN {X 0,Y 303.605,Z 720.168,A -85,B 0,C 180,E1 -16126.126,E2 -16126.126} C_VEL
LIN {X 0,Y 303.787,Z 719.611,A -85,B 0,C 180,E1 -16128.896,E2 -16128.896} C_VEL
LIN {X 0,Y 304.14,Z 718.037,A -85,B 0,C 180,E1 -16131.697,E2 -16131.697} C_VEL
LIN {X 0,Y 304.8,Z 715.424,A -85,B 0,C 180,E1 -16134.52,E2 -16134.52} C_VEL
LIN {X 0,Y 305.841,Z 711.586,A -85,B 0,C 180,E1 -16137.358,E2 -16137.358} C_VEL
LIN {X 0,Y 307.205,Z 706.554,A -85,B 0,C 180,E1 -16140.216,E2 -16140.216} C_VEL
LIN {X 0,Y 309.081,Z 700.192,A -85,B 0,C 180,E1 -16143.072,E2 -16143.072} C_VEL
LIN {X 0,Y 311.554,Z 692.274,A -85,B 0,C 180,E1 -16145.907,E2 -16145.907} C_VEL
LIN {X 0,Y 314.664,Z 682.591,A -85,B 0,C 180,E1 -16148.708,E2 -16148.708} C_VEL
LIN {X 0,Y 317.909,Z 672.312,A -85,B 0,C 180,E1 -16151.147,E2 -16151.147} C_VEL
LIN {X 0,Y 320.887,Z 662.34,A -85,B 0,C 180,E1 -16153.147,E2 -16153.147} C_VEL
LIN {X 0,Y 324.458,Z 650.21,A -85,B 0,C 180,E1 -16155.183,E2 -16155.183} C_VEL
LIN {X 0,Y 327.923,Z 637.234,A -85,B 0,C 180,E1 -16156.998,E2 -16156.998} C_VEL
LIN {X 0,Y 331.241,Z 623.433,A -85,B 0,C 180,E1 -16158.588,E2 -16158.588} C_VEL
LIN {X 0,Y 334.118,Z 609.585,A -85,B 0,C 180,E1 -16159.916,E2 -16159.916} C_VEL
LIN {X 0,Y 336.366,Z 597.673,A -85,B 0,C 180,E1 -16160.862,E2 -16160.862} C_VEL
LIN {X 0,Y 334.261,Z 588.612,A -85,B 0,C 180,E1 -16162.032,E2 -16162.032} C_VEL
LIN {X 0,Y 330.128,Z 576.093,A -85,B 0,C 180,E1 -16163.694,E2 -16163.694} C_VEL
LIN {X 0,Y 329.091,Z 573.429,A -85,B 0,C 180,E1 -16164.064,E2 -16164.064} C_VEL
LIN {X 0,Y 327.481,Z 570.929,A -85,B 0,C 180,E1 -16164.526,E2 -16164.526} C_VEL
LIN {X 0,Y 323.652,Z 568.307,A -85,B 0,C 180,E1 -16165.397,E2 -16165.397} C_VEL
LIN {X 0,Y 319.799,Z 565.645,A -85,B 0,C 180,E1 -16166.271,E2 -16166.271} C_VEL
LIN {X 0,Y 318.133,Z 563.085,A -85,B 0,C 180,E1 -16166.729,E2 -16166.729} C_VEL
LIN {X 0,Y 312.899,Z 553.673,A -85,B 0,C 180,E1 -16168.28,E2 -16168.28} C_VEL
LIN {X 0,Y 310.392,Z 549.725,A -85,B 0,C 180,E1 -16168.983,E2 -16168.983} C_VEL
LIN {X 0,Y 308.038,Z 546.028,A -85,B 0,C 180,E1 -16169.658,E2 -16169.658} C_VEL
LIN {X 0,Y 305.5,Z 542.264,A -85,B 0,C 180,E1 -16170.369,E2 -16170.369} C_VEL
LIN {X 0,Y 302.475,Z 538.323,A -85,B 0,C 180,E1 -16171.222,E2 -16171.222} C_VEL
LIN {X 0,Y 301.769,Z 536.613,A -85,B 0,C 180,E1 -16171.482,E2 -16171.482} C_VEL
LIN {X 0,Y 301.042,Z 532.518,A -85,B 0,C 180,E1 -16175.151,E2 -16175.151} C_VEL
LIN {X 0,Y 300.422,Z 529.508,A -85,B 0,C 180,E1 -16178.018,E2 -16178.018} C_VEL
LIN {X 0,Y 299.792,Z 526.575,A -85,B 0,C 180,E1 -16180.84,E2 -16180.84} C_VEL
LIN {X 0,Y 298.75,Z 522.483,A -85,B 0,C 180,E1 -16185.002,E2 -16185.002} C_VEL
LIN {X 0,Y 298.567,Z 521.599,A -85,B 0,C 180,E1 -16186.038,E2 -16186.038} C_VEL
LIN {X 0,Y 298.751,Z 521.579,A -85,B 0,C 180,E1 -16191.113,E2 -16191.113} C_VEL
LIN {X 0,Y 298.79,Z 521.578,A -85,B 0,C 180,E1 -16193.245,E2 -16193.245} C_VEL
LIN {X 0,Y 298.839,Z 521.57,A -85,B 0,C 180,E1 -16197.303,E2 -16197.303} C_VEL
LIN {X 0,Y 299.016,Z 521.552,A -85,B 0,C 180,E1 -16199.999,E2 -16199.999} C_VEL
LIN {X 0,Y 298.828,Z 521.565,A -85,B 0,C 180,E1 -16202.695,E2 -16202.695} C_VEL
LIN {X 0,Y 298.787,Z 521.575,A -85,B 0,C 180,E1 -16206.754,E2 -16206.754} C_VEL
LIN {X 0,Y 298.67,Z 521.581,A -85,B 0,C 180,E1 -16209.48,E2 -16209.48} C_VEL
LIN {X 0,Y 298.543,Z 521.603,A -85,B 0,C 180,E1 -16213.615,E2 -16213.615} C_VEL
LIN {X 0,Y 298.538,Z 521.566,A -85,B 0,C 180,E1 -16216.409,E2 -16216.409} C_VEL
LIN {X 0,Y 298.555,Z 521.577,A -85,B 0,C 180,E1 -16219.684,E2 -16219.684} C_VEL
LIN {X 0,Y 298.478,Z 521.573,A -85,B 0,C 180,E1 -16223.595,E2 -16223.595} C_VEL
LIN {X 0,Y 298.479,Z 521.591,A -85,B 0,C 180,E1 -16226.575,E2 -16226.575} C_VEL
LIN {X 0,Y 298.471,Z 521.765,A -85,B 0,C 180,E1 -16229.025,E2 -16229.025} C_VEL
LIN {X 0,Y 300.201,Z 529.679,A -85,B 0,C 180,E1 -16233.377,E2 -16233.377} C_VEL
LIN {X 0,Y 301.808,Z 537.172,A -85,B 0,C 180,E1 -16237.26,E2 -16237.26} C_VEL
LIN {X 0,Y 303.216,Z 543.661,A -85,B 0,C 180,E1 -16240.465,E2 -16240.465} C_VEL
LIN {X 0,Y 305.009,Z 552.456,A -85,B 0,C 180,E1 -16244.544,E2 -16244.544} C_VEL
LIN {X 0,Y 305.422,Z 554.176,A -85,B 0,C 180,E1 -16244.941,E2 -16244.941} C_VEL
LIN {X 0,Y 307.413,Z 558.323,A -85,B 0,C 180,E1 -16245.528,E2 -16245.528} C_VEL
LIN {X 0,Y 308.935,Z 560.735,A -85,B 0,C 180,E1 -16245.94,E2 -16245.94} C_VEL
LIN {X 0,Y 311.635,Z 566.933,A -85,B 0,C 180,E1 -16246.719,E2 -16246.719} C_VEL
LIN {X 0,Y 316.525,Z 581.689,A -85,B 0,C 180,E1 -16248.235,E2 -16248.235} C_VEL
LIN {X 0,Y 320.561,Z 597.377,A -85,B 0,C 180,E1 -16249.808,E2 -16249.808} C_VEL
LIN {X 0,Y 322.638,Z 608.962,A -85,B 0,C 180,E1 -16250.94,E2 -16250.94} C_VEL
LIN {X 0,Y 324.442,Z 624.698,A -85,B 0,C 180,E1 -16252.537,E2 -16252.537} C_VEL
LIN {X 0,Y 325.371,Z 639.901,A -85,B 0,C 180,E1 -16254.204,E2 -16254.204} C_VEL
LIN {X 0,Y 323.153,Z 650.851,A -85,B 0,C 180,E1 -16255.19,E2 -16255.19} C_VEL
LIN {X 0,Y 319.67,Z 664.958,A -85,B 0,C 180,E1 -16256.66,E2 -16256.66} C_VEL
LIN {X 0,Y 315.951,Z 679.176,A -85,B 0,C 180,E1 -16258.486,E2 -16258.486} C_VEL
LIN {X 0,Y 312.611,Z 691.284,A -85,B 0,C 180,E1 -16260.359,E2 -16260.359} C_VEL
LIN {X 0,Y 309.038,Z 703.442,A -85,B 0,C 180,E1 -16262.615,E2 -16262.615} C_VEL
LIN {X 0,Y 306.027,Z 713.597,A -85,B 0,C 180,E1 -16264.86,E2 -16264.86} C_VEL
LIN {X 0,Y 303.147,Z 723.657,A -85,B 0,C 180,E1 -16267.512,E2 -16267.512} C_VEL
LIN {X 0,Y 300.926,Z 732.163,A -85,B 0,C 180,E1 -16270.208,E2 -16270.208} C_VEL
LIN {X 0,Y 298.826,Z 740.81,A -85,B 0,C 180,E1 -16273.609,E2 -16273.609} C_VEL
LIN {X 0,Y 297.763,Z 746.336,A -85,B 0,C 180,E1 -16276.35,E2 -16276.35} C_VEL
LIN {X 0,Y 297.025,Z 750.782,A -85,B 0,C 180,E1 -16279.09,E2 -16279.09} C_VEL
LIN {X 0,Y 296.784,Z 754.161,A -85,B 0,C 180,E1 -16281.833,E2 -16281.833} C_VEL
LIN {X 0,Y 296.754,Z 756.51,A -85,B 0,C 180,E1 -16284.566,E2 -16284.566} C_VEL
LIN {X 0,Y 296.749,Z 757.867,A -85,B 0,C 180,E1 -16287.287,E2 -16287.287} C_VEL
LIN {X 0,Y 296.99,Z 758.219,A -85,B 0,C 180,E1 -16290.001,E2 -16290.001} C_VEL
LIN {X 0,Y 296.799,Z 757.561,A -85,B 0,C 180,E1 -16292.716,E2 -16292.716} C_VEL
LIN {X 0,Y 296.867,Z 755.286,A -85,B 0,C 180,E1 -16296.123,E2 -16296.123} C_VEL
LIN {X 0,Y 296.821,Z 753.157,A -85,B 0,C 180,E1 -16298.169,E2 -16298.169} C_VEL
LIN {X 0,Y 297.071,Z 749.301,A -85,B 0,C 180,E1 -16300.911,E2 -16300.911} C_VEL
LIN {X 0,Y 297.763,Z 744.386,A -85,B 0,C 180,E1 -16303.653,E2 -16303.653} C_VEL
LIN {X 0,Y 298.759,Z 738.173,A -85,B 0,C 180,E1 -16306.398,E2 -16306.398} C_VEL
LIN {X 0,Y 300.345,Z 730.636,A -85,B 0,C 180,E1 -16309.124,E2 -16309.124} C_VEL
LIN {X 0,Y 302.287,Z 721.587,A -85,B 0,C 180,E1 -16311.84,E2 -16311.84} C_VEL
LIN {X 0,Y 304.546,Z 712.268,A -85,B 0,C 180,E1 -16314.182,E2 -16314.182} C_VEL
LIN {X 0,Y 312.16,Z 685.514,A -85,B 0,C 180,E1 -16319.691,E2 -16319.691} C_VEL
LIN {X 0,Y 317.416,Z 669.958,A -85,B 0,C 180,E1 -16322.334,E2 -16322.334} C_VEL
LIN {X 0,Y 323.083,Z 653.773,A -85,B 0,C 180,E1 -16324.633,E2 -16324.633} C_VEL
LIN {X 0,Y 327.141,Z 642.297,A -85,B 0,C 180,E1 -16326.023,E2 -16326.023} C_VEL
LIN {X 0,Y 329.27,Z 629.622,A -85,B 0,C 180,E1 -16327.941,E2 -16327.941} C_VEL
LIN {X 0,Y 331.885,Z 616.792,A -85,B 0,C 180,E1 -16329.788,E2 -16329.788} C_VEL
LIN {X 0,Y 333.528,Z 606.223,A -85,B 0,C 180,E1 -16331.569,E2 -16331.569} C_VEL
LIN {X 0,Y 334.774,Z 597.615,A -85,B 0,C 180,E1 -16333.326,E2 -16333.326} C_VEL
LIN {X 0,Y 335.913,Z 591.42,A -85,B 0,C 180,E1 -16334.93,E2 -16334.93} C_VEL
LIN {X 0,Y 336.187,Z 590.191,A -85,B 0,C 180,E1 -16335.299,E2 -16335.299} C_VEL
LIN {X 0,Y 336.525,Z 588.008,A -85,B 0,C 180,E1 -16336.436,E2 -16336.436} C_VEL
LIN {X 0,Y 337.36,Z 586.073,A -85,B 0,C 180,E1 -16338.193,E2 -16338.193} C_VEL
LIN {X 0,Y 338.614,Z 585.867,A -85,B 0,C 180,E1 -16340.171,E2 -16340.171} C_VEL
LIN {X 0,Y 340.034,Z 586.966,A -85,B 0,C 180,E1 -16341.759,E2 -16341.759} C_VEL
LIN {X 0,Y 341.261,Z 588.835,A -85,B 0,C 180,E1 -16343.01,E2 -16343.01} C_VEL
LIN {X 0,Y 334.713,Z 605.845,A -85,B 0,C 180,E1 -16345.062,E2 -16345.062} C_VEL
LIN {X 0,Y 328.88,Z 620.308,A -85,B 0,C 180,E1 -16347.174,E2 -16347.174} C_VEL
LIN {X 0,Y 323.652,Z 632.76,A -85,B 0,C 180,E1 -16349.317,E2 -16349.317} C_VEL
LIN {X 0,Y 318.644,Z 644.603,A -85,B 0,C 180,E1 -16351.765,E2 -16351.765} C_VEL
LIN {X 0,Y 313.941,Z 655.478,A -85,B 0,C 180,E1 -16354.474,E2 -16354.474} C_VEL
LIN {X 0,Y 310.662,Z 662.885,A -85,B 0,C 180,E1 -16356.679,E2 -16356.679} C_VEL
LIN {X 0,Y 307.513,Z 670.18,A -85,B 0,C 180,E1 -16359.254,E2 -16359.254} C_VEL
LIN {X 0,Y 304.838,Z 676.332,A -85,B 0,C 180,E1 -16361.867,E2 -16361.867} C_VEL
LIN {X 0,Y 302.624,Z 681.318,A -85,B 0,C 180,E1 -16364.511,E2 -16364.511} C_VEL
LIN {X 0,Y 301.359,Z 684.392,A -85,B 0,C 180,E1 -16366.514,E2 -16366.514} C_VEL
LIN {X 0,Y 299.646,Z 688.382,A -85,B 0,C 180,E1 -16370.095,E2 -16370.095} C_VEL
LIN {X 0,Y 298.666,Z 690.48,A -85,B 0,C 180,E1 -16373.244,E2 -16373.244} C_VEL
LIN {X 0,Y 297.97,Z 691.218,A -85,B 0,C 180,E1 -16375.943,E2 -16375.943} C_VEL
LIN {X 0,Y 297.52,Z 691.069,A -85,B 0,C 180,E1 -16378.647,E2 -16378.647} C_VEL
LIN {X 0,Y 297.487,Z 689.86,A -85,B 0,C 180,E1 -16381.354,E2 -16381.354} C_VEL
LIN {X 0,Y 297.774,Z 687.694,A -85,B 0,C 180,E1 -16384.061,E2 -16384.061} C_VEL
LIN {X 0,Y 297.817,Z 684.545,A -85,B 0,C 180,E1 -16386.777,E2 -16386.777} C_VEL
LIN {X 0,Y 298.314,Z 680.276,A -85,B 0,C 180,E1 -16389.493,E2 -16389.493} C_VEL
LIN {X 0,Y 298.935,Z 674.912,A -85,B 0,C 180,E1 -16392.216,E2 -16392.216} C_VEL
LIN {X 0,Y 300.021,Z 668.285,A -85,B 0,C 180,E1 -16394.933,E2 -16394.933} C_VEL
LIN {X 0,Y 301.435,Z 660.26,A -85,B 0,C 180,E1 -16397.644,E2 -16397.644} C_VEL
LIN {X 0,Y 303.267,Z 650.699,A -85,B 0,C 180,E1 -16400.342,E2 -16400.342} C_VEL
LIN {X 0,Y 305.338,Z 640.27,A -85,B 0,C 180,E1 -16402.819,E2 -16402.819} C_VEL
LIN {X 0,Y 307.514,Z 629.448,A -85,B 0,C 180,E1 -16405.012,E2 -16405.012} C_VEL
LIN {X 0,Y 310.288,Z 616.008,A -85,B 0,C 180,E1 -16407.301,E2 -16407.301} C_VEL
LIN {X 0,Y 313.135,Z 601.264,A -85,B 0,C 180,E1 -16409.404,E2 -16409.404} C_VEL
LIN {X 0,Y 315.716,Z 586.474,A -85,B 0,C 180,E1 -16411.169,E2 -16411.169} C_VEL
LIN {X 0,Y 318.147,Z 572.085,A -85,B 0,C 180,E1 -16412.593,E2 -16412.593} C_VEL
LIN {X 0,Y 318.395,Z 570.2,A -85,B 0,C 180,E1 -16412.773,E2 -16412.773} C_VEL
LIN {X 0,Y 317.276,Z 566.384,A -85,B 0,C 180,E1 -16413.258,E2 -16413.258} C_VEL
